// Set Control Mode Label
CASE stat.nCtrlMode	OF
	0:	stat.sCtrlMode	:= 'HHR (Hand-Held Remote)';
	1:	stat.sCtrlMode	:= 'REMOTE';
	2:	stat.sCtrlMode	:= 'SERIAL LINK';
	3:	stat.sCtrlMode	:= 'FIELDBUS';
ELSE
	stat.sCtrlMode	:= 'UNKNOWN';
END_CASE
END_METHOD

END_FUNCTION_BLOCK

// POUs/Pumps/FB_CRYO_PUMP_SERIAL
// Cryo Turbo Molecular Pump Control
FUNCTION_BLOCK FB_CRYO_PUMP_SERIAL EXTENDS FB_CRYO_PUMP_BASE
VAR_INPUT
	{attribute 'OPC.UA.DA' := '0'}
	in_sCmdSuffix:		STRING(16) := '$0D';
	{attribute 'OPC.UA.DA' := '0'}
	in_sReplySuffix:	STRING(16) := '$0D';
END_VAR
VAR_OUTPUT
END_VAR
VAR

	{attribute 'OPC.UA.DA' := '0'}
	comm:		FB_RS_COMM_NO_SIM;			// No simulation yet
	
	// Pointers to structures inside FB_RS_COMM, e.g. ptrCommCfg.
	{attribute 'OPC.UA.DA' := '0'}
	ptrCommCfg:		POINTER TO T_RS_COMM_CFG;	(* Pointer to comm.cfg instance *)
	{attribute 'OPC.UA.DA' := '0'}
	ptrCommCtrl:	POINTER TO T_RS_COMM_CTRL;	(* Pointer to comm.ctrl instance *)
	{attribute 'OPC.UA.DA' := '0'}
	ptrCommStat:	POINTER TO T_RS_COMM_STAT;	(* Pointer to comm.stat instance *)

END_VAR

// Execute the base class object FB_RS_BASE
SUPER^();

METHOD ActivityInitializing
VAR_INPUT
	bExecute:	BOOL;
END_VAR
VAR_INST
	{attribute 'OPC.UA.DA' := '0'}
    nMethodState:	INT := 0;	// State Machine current state
END_VAR
SetAction('ActivityInitializing');


IF NOT bExecute THEN
	nMethodState	:= 0;	// Reset the state machine
	cmdCounter		:= 0;	// Init will start from the first init command after increment
	RETURN;
END_IF

// Handle State Machine
CASE nMethodState OF
	0:	// Set initial state and status
		statRef.bInitialised	:= FALSE;
		statBaseRef.sReply			:= '';
		SetStatus(E_SM_ERROR.OK, 'BUSY');

		nMethodState := 10;				// Go to next state, i.e. INIT_COMM

	10:	// Initialize COMM port
		(* Reset the serial port *)
		ptrCommCtrl^.nCommand	:= E_RS_COMM_CMD.INIT;
		ptrCommCtrl^.bExecute	:= TRUE;

		(* Start the timer by going false/true *)
		fbTimer (IN := FALSE); (* Reset timer *)
		fbTimer (IN := TRUE, PT := T#5S); (* 5 sec timeout for reply *)

		nMethodState 	:= 15;	// On next cycle wait until the comm port is reset, i.e. idle
		
	15:	// Wait IDLE
		fbTimer (IN := TRUE);
		IF comm.stat.nStatus = E_RS_COMM_STATUS.IDLE THEN
			// Communication is IDLE 
			fbTimer (IN := FALSE);	// disable timer 
			statBaseRef.sReply		:= ptrCommStat^.sReply;	// Save the reply

			// TODO Assign the value to a status variable.
			IF NOT M_ReadFromReply(cmdCounter, TRUE)	THEN
				cmdCounter		:= 0;	// Reset command counter
				nMethodState 	:= 10;	// Wait for INIT
			ELSE
				cmdCounter		:= cmdCounter + 1;	// Increment init command index
				fbTimer (IN := FALSE);	// disable timer 
				fbTimer (IN := TRUE, PT := cfgRef.tDelay_Init); // Wait INIT delay
				bCommProblem	:= FALSE;
				nMethodState 	:= 18;	// Execute next device INIT command
			END_IF
		ELSIF comm.stat.nStatus = E_RS_COMM_STATUS.ERROR THEN
			fbTimer (IN := FALSE);
			SetStatus(E_LAKESHORE_ERROR.COMM, 'ERROR: Communication error');	
			bCommProblem	:= TRUE;
			nEvent := E_SM_EVENT.ERRINIT;
			RETURN;
		ELSIF fbTimer.Q THEN
			// Timer expired after 5 sec. This is an error.
			fbTimer (IN := FALSE);
			SetStatus(E_LAKESHORE_ERROR.TIMEOUT, 'ERROR: Communication timeout');	
			bCommProblem	:= TRUE;
			nEvent := E_SM_EVENT.ERRINIT;
			RETURN;
		END_IF

	
	
	18:	// Wait INIT Delay
		fbTimer (IN := TRUE);
		IF fbTimer.Q THEN
			// Timer expired after 5 sec. This is an error.
			fbTimer (IN := FALSE);
			nMethodState 	:= 20;	// Execute next device INIT command
			RETURN;
		END_IF

	
	
	20:	// INIT DEV
		IF ptrInitCmds^ [cmdCounter].cmd = '' THEN
			// Device INIT is done. Go to IDLE 
			statRef.bInitialised 	:= TRUE;
			cmdCounter			:= 1;
			SetStatus(E_SM_ERROR.OK, 'IDLE');
			nEvent 		:= E_SM_EVENT.INITDONE;
			RETURN;
		END_IF
		
		(* Send INIT command with index cmdCounter *)
		ptrCommCtrl^.nCommand		:= E_RS_COMM_CMD.SEND;
		ptrCommCtrl^.sCmd			:= ptrInitCmds^ [cmdCounter].cmd;
		ptrCommCtrl^.nNumReplies	:= 1;
		ptrCommCtrl^.bHasReply		:= TRUE;
		ptrCommCtrl^.bExecute		:= TRUE;
	
		(* Start the timer by going false/true *)
		fbTimer (IN := FALSE); (* Reset timer *)
		fbTimer (IN := TRUE, PT := T#5S); (* 5 sec timeout for reply *)

		// On next cycle wait until the comm port is idle
		nMethodState 	:= 15;	// On next cycle wait until the comm port is idle
	
END_CASE
END_METHOD

METHOD ActivityMonitoring
VAR_INPUT
	bExecute:	BOOL;
END_VAR
VAR_INST
	{attribute 'OPC.UA.DA' := '0'}
    nMethodState:	INT := 0;	// State Machine current state
	{attribute 'OPC.UA.DA' := '0'}
	nRetries:		INT := 0;	// Number of retries in case of communication problems
END_VAR

VAR
	offset: INT;
END_VAR
IF NOT cfgRef.bAutoMonitor AND statRef.nSubstate = E_RS_BASE_SUBSTATE.NOTOP_READY THEN
	SetAction('No Monitoring'); 
	SetStatus(E_SM_ERROR.OK, 'IDLE');
	nMethodState	:= 0;	// Reset the state machine
	cmdCounter		:= 1;	// Reading will start from the first command in the array
	RETURN;
END_IF

IF NOT bExecute THEN
	SetAction('ActivityMonitoring'); 
	SetStatus(E_SM_ERROR.OK, 'BUSY');
	nMethodState	:= 0;	// Reset the state machine
	cmdCounter		:= 1;	// Reading will start from the first command in the array
	RETURN;
END_IF

// Handle State Machine
CASE nMethodState OF
	0:	// Execute a command from the command array
		IF ptrReadCmds^ [cmdCounter].cmd = '' OR cmdCounter > 16 THEN

			// All commands have been executed. 
			// Wait tDelay_Periodic before re-starting the READ.
			cmdCounter	:= 1;
			SetStatus(E_SM_ERROR.OK, 'IDLE');
			
			(* Start the timer by going false/true *)
			fbTimer (IN := FALSE); (* Reset timer *)
			fbTimer (IN := TRUE, PT := cfgRef.tDelay_Periodic);
			nMethodState := 10;				// Goto Wait for tDelay_Periodic
			RETURN;
			
		END_IF
		
		(* Send command with index cmdCounter *)
		ptrCommCtrl^.nCommand		:= E_RS_COMM_CMD.SEND;
		ptrCommCtrl^.sCmd			:= ptrReadCmds^ [cmdCounter].cmd;
		ptrCommCtrl^.nNumReplies	:= 1;
		ptrCommCtrl^.bHasReply		:= TRUE;
		ptrCommCtrl^.bExecute		:= TRUE;
		
		// In case we are executing 'SET' commands, there are no replies.
		// However, we need a delay of at least 50ms between commands.
		// We will apply 150ms.
		IF NOT ptrCommCtrl^.bHasReply THEN
			// There is no reply, i.e. this is a 'SET' command.
			// Start the timer by going false/true.
			// Apply 200ms delay between SET commands.
			fbTimer (IN := FALSE); // Reset timer
			fbTimer (IN := TRUE, PT := T#200MS); 
			cmdCounter		:= cmdCounter + 1;	// Go to next command.
			nMethodState	:= 10;				// Goto WAIT for Reading to complete,
			RETURN;
		ELSE			
			// There is a reply, i.e. this is a 'READ' command.
			// Apply short delay of 10ms before checking the status. 
			// Start the timer by going false/true
			fbTimer (IN := FALSE); // Reset timer
			fbTimer (IN := TRUE, PT := T#10MS);	
			statRef.sErrorText	:= 'BUSY';
			nMethodState := 15;	// Goto WAIT for Reading to complete,
		END_IF
		

	10:	// Wait until the delay timeout expires
		fbTimer (IN := TRUE);

		(* If Timer has expired, go to the next state. *)
		IF fbTimer.Q THEN
			fbTimer (IN := FALSE);
			nMethodState 	:= 0;	// Goto Wait for tDelay_Periodic
			RETURN;
		END_IF
	
	15:	// Wait until the delay timeout expires
		fbTimer (IN := TRUE);

		(* If Timer has expired, go to the next state. *)
		IF fbTimer.Q THEN
			fbTimer (IN := FALSE);
			fbTimer (IN := TRUE, PT := T#5S);	// 5 sec timeout for reply
			statRef.sErrorText	:= 'BUSY';
			nMethodState 	:= 20;	// Goto Wait for IDLE/Reply
			RETURN;
		END_IF
	



	20:	// Wait for the reading to complete, i.e. IDLE
		fbTimer (IN := TRUE);
		IF comm.stat.nStatus = E_RS_COMM_STATUS.IDLE THEN
			// Communication is IDLE 
			fbTimer (IN := FALSE);	// disable timer 
			statBaseRef.sReply		:= ptrCommStat^.sReply;	// Save the reply
			
			// Copy readings to status variable(s)
			
			// TODO Assign the value to a status variable.
			IF NOT M_ReadFromReply(cmdCounter, FALSE)	THEN
				// Reply was not OK. Maybe out of sync.
				// Re-INIT the communication, i.e. clear the buffer.
				ptrCommCtrl^.nCommand	:= E_RS_COMM_CMD.INIT;
				ptrCommCtrl^.bExecute	:= TRUE;
		
				(* Start the timer by going false/true *)
				fbTimer (IN := FALSE); (* Reset timer *)
				fbTimer (IN := TRUE, PT := T#5S); (* 5 sec timeout for reply *)
		
				SetStatus(E_LAKESHORE_ERROR.COMM, 'ERROR: Communication error');	
				bCommProblem	:= TRUE;

				nMethodState 	:= 10;	// On next cycle wait until the comm port is reset, i.e. idle
				RETURN;
			ELSE
				// All OK. Go to next command.
				bCommProblem	:= FALSE;
				nRetries		:= 0;	// Reset number of retries
		
				cmdCounter		:= cmdCounter + 1;	// Go to next command.
				
				// Apply a 50 ms delay between commands
				fbTimer (IN := FALSE);	// Reset timer
				fbTimer (IN := TRUE, PT := T#50MS); 
				nMethodState := 10;		// Apply delay
				nEvent := E_SM_EVENT.COMMOK;
				RETURN;
			END_IF
		ELSIF comm.stat.nStatus = E_RS_COMM_STATUS.ERROR OR fbTimer.Q THEN
			// No Reply.
			// Re-INIT the communication, i.e. clear the buffer.
			ptrCommCtrl^.nCommand	:= E_RS_COMM_CMD.INIT;
			ptrCommCtrl^.bExecute	:= TRUE;
	
			(* Start the timer by going false/true *)
			fbTimer (IN := FALSE); (* Reset timer *)
			fbTimer (IN := TRUE, PT := T#5S); (* 5 sec timeout for reply *)
	
			SetStatus(E_LAKESHORE_ERROR.COMM, 'ERROR: Communication error');	
			bCommProblem	:= TRUE;

			nRetries		:= nRetries + 1;		// Increment number of retries
			statBaseRef.nRetries	:= statBaseRef.nRetries + 1;	// Increment total number of retries

			nMethodState 	:= 10;	// On next cycle wait until the comm port is reset, i.e. idle
			RETURN;
		END_IF

	
END_CASE
END_METHOD

METHOD M_ExecuteComm
VAR_INPUT
END_VAR
comm(in_sCmdSuffix:=in_sCmdSuffix, in_sReplySuffix:=in_sReplySuffix, in_nTimeout:=3000);
END_METHOD

METHOD M_GetCouplerState : BOOL
VAR_INPUT
END_VAR
IF comm.i_nCouplerState = 8 THEN
	M_GetCouplerState	:= TRUE;	
ELSE
	M_GetCouplerState	:= FALSE;	
END_IF
END_METHOD

// Add checksum at the end of Pfeiffer Vacuum Protocol (PVP) command
METHOD M_PVP_Checksum : STRING(24)
VAR_INPUT
	sCmd:	STRING;	// Command without the checksum
END_VAR
VAR
	i:			INT;
	nVar:		SINT;
	nSum:		INT;
	nRes:		INT;	// Resulting check sum
	sCmdFull:	STRING(24);	// Command with the checksum
    fbFormat:	FB_FormatString;
	sTmp:		T_MaxString;
	length:		INT;
END_VAR
// Get the command length
length	:= LEN(sCmd);

nSum	:= 0;
FOR i:=0 TO (length-1) DO
	nSum	:= nSum + BYTE_TO_SINT(sCmd[i]);
END_FOR
nRes	:= nSum MOD 256;

sTmp	:= sCmd;
fbFormat(	sFormat := '%s%.3d', 
			arg1 := F_STRING(sTmp), 
			arg2 := F_INT(nRes), 
			sOut => sCmdFull);
			
M_PVP_Checksum	:= sCmdFull;
END_METHOD

METHOD M_ReadFromReply : BOOL
// Method to check correctness of the reply and assign the result to a status variable.
VAR_INPUT
	idx:		INT;		(* arr [idx] will hold the first extracted value, arr [idx+1] the second one, etc. *)
	bInitCmd:	BOOL := FALSE;
END_VAR
VAR
	pos:	INT;
	cmd:	STRING;
	length:	DINT;
	subStr:	STRING(255);
END_VAR
// TODO: Implement specific parsing of replies
END_METHOD

END_FUNCTION_BLOCK

// POUs/Pumps/FB_CRYO_PUMP_ECODRY
FUNCTION_BLOCK FB_CRYO_PUMP_ECODRY EXTENDS FB_CRYO_PUMP_MODBUS
VAR_INPUT
END_VAR
VAR_OUTPUT
END_VAR
VAR CONSTANT
END_VAR
VAR
	{attribute 'OPC.UA.DA' := '1'}
	cfg:		T_CRYO_PUMP_MODBUS_CFG;		//  Config parameters
	{attribute 'OPC.UA.DA' := '1'}
	ctrl:		T_CRYO_PUMP_MODBUS_CTRL;	//  Control parameters
	{attribute 'OPC.UA.DA' := '1'}
	{attribute 'OPC.UA.DA.Access' := '1'}
	stat:		T_CRYO_PUMP_MODBUS_STAT;	//  Status parameters - ReadOnly


END_VAR

// Execute the base class object FB_RS_BASE
SUPER^();

METHOD M_Configure
VAR_INPUT
END_VAR
IF NOT bStarted	THEN
	//
	// START: Mandatory for ALL pumps !!!
	//
	// Set references from FB_RS_BASE
	cfgRef	REF=cfg;
	ctrlRef	REF=ctrl;
	statRef	REF=stat;

	// Set references from FB_CRYO_PUMP_BASE
	cfgBaseRef	REF=cfg;
	ctrlBaseRef	REF=ctrl;
	statBaseRef	REF=stat;

	// Set references from FB_CRYO_PUMP_MODBUS
	cfgModbusRef	REF=cfg;
	ctrlModbusRef	REF=ctrl;
	statModbusRef	REF=stat;

	// Copy input parameters to configuration
	cfg.nModel			:= in_nModel;
	cfg.bAutoMonitor	:= in_bAutoMonitor;
	cfg.tDelay_Periodic	:= DINT_TO_TIME(in_nPeriod);
	
	
	// Set pointers to arrays of commands
//	ptrInitCmds	:= ADR(cfg.cmdList_Init);(* Pointer to INIT commands *)
//	ptrReadCmds	:= ADR(cfg.cmdList_Read);(* Pointer to READ commands *)
	
	// TODO in FB that extends the functionality
	// Set pointers to comm, i.e.
	ptrCommCfg	:= ADR(comm.cfg);	(* Pointer to comm.cfg instance *)
	ptrCommCtrl	:= ADR(comm.ctrl);	(* Pointer to comm.ctrl instance *)
	ptrCommStat	:= ADR(comm.stat);	(* Pointer to comm.stat instance *)
	
	// Set comm suffixes for commands and replies
//	ptrCommCfg^.sCmdSuffix		:= '';
//	ptrCommCfg^.sReplySuffix	:= '';

	statRef.bConfigured	:= TRUE;
	bStarted			:= TRUE;
	//
	// END: Mandatory for ALL pumps !!!
	//


	// TODO USER
	// Add here real configuration
	IF in_sVersion = 'V01'	THEN
		cfg.nVersion	:= E_ECODRY_VERSION.V01;
	ELSIF in_sVersion = 'V21'  OR  in_sVersion = 'V22'	THEN
		cfg.nVersion	:= E_ECODRY_VERSION.V21_22;
	END_IF
	
	// Adjust addresses and number of words
	CASE cfg.nVersion	OF
		E_ECODRY_VERSION.V01:
			// Set register addresses
			cfg.aAddr [1]	:= 16#0040;
			cfg.aAddr [2]	:= 16#0067;
			cfg.aAddr [3]	:= 16#0667;
			cfg.aAddr [4]	:= 0;	// Unused address must be zero
			
			// Set number of words to read
			cfg.aWords [1]	:= 16;
			cfg.aWords [2]	:= 2;
			cfg.aWords [3]	:= 6;
			cfg.aWords [4]	:= 0;	// Number of words for unused address must be zero
	END_CASE
	
	cfg.nSlaveID	:= in_nSlaveID;

	
END_IF
END_METHOD

METHOD M_ExtractReadings_V01 : BOOL
VAR_INPUT
	nAddressIndex:	INT;	// Which address space to read
END_VAR
VAR
	pBuf:	POINTER TO BYTE	:= ADR(stat.nInputBuffer);
	loop:	INT;
	par:	INT;
END_VAR
// There are 3 bytes before data starts !!!
IF nAddressIndex = 1 THEN
	////////////////////////////
	// Extract Common Parameters
	////////////////////////////

	// Reference Frequency 0x40H
	// Offset 3 + 0 = 3
	stat.lrFreqRef		:= UINT_TO_LREAL(M_ByteSwapUINT(ADR(pBuf[3]))) / 100.0;
	stat.lrOutFreq		:= INT_TO_LREAL(M_ByteSwapINT(ADR(pBuf[5]))) / 100.0;
	stat.nPumpSpeed		:= LREAL_TO_DINT(stat.lrOutFreq * 60.0);	// [Hz] -> [rpm]
	stat.nMotorCurr		:= UINT_TO_DINT(M_ByteSwapUINT(ADR(pBuf[7]))) * 10;
	stat.lrOutVoltRef	:= UINT_TO_LREAL(M_ByteSwapUINT(ADR(pBuf[13]))) / 10.0;
	stat.nMotorVolt		:= UINT_TO_DINT(M_ByteSwapUINT(ADR(pBuf[15])));
	stat.lrOutPower		:= INT_TO_LREAL(M_ByteSwapINT(ADR(pBuf[17]))) / 10.0;
	
	stat.nOpTime	:= M_ByteSwapUINT(ADR(pBuf[27]));
	stat.nSwFlash	:= M_ByteSwapUINT(ADR(pBuf[29]));

	(*
	stat.lrTemperature	:= UINT_TO_LREAL(M_ByteSwapUINT(ADR(pBuf[83])));

	stat.nSwRom		:= M_ByteSwapUINT(ADR(pBuf[57]));
	stat.nNumRunCmd	:= M_ByteSwapUINT(ADR(pBuf[109]));
	stat.nFanOpTime	:= M_ByteSwapUINT(ADR(pBuf[81]));
	*)

ELSIF nAddressIndex = 2 THEN
	stat.nFanOpTime			:= M_ByteSwapUINT(ADR(pBuf[3]));
	stat.nElecTemp			:= UINT_TO_DINT(M_ByteSwapUINT(ADR(pBuf[5])));
ELSIF nAddressIndex = 3 THEN
	stat.nServiceHours		:= M_ByteSwapUINT(ADR(pBuf[3]));
	stat.nNumPumpDowns		:= M_ByteSwapUINT(ADR(pBuf[7]));
	stat.nDaysUntilService	:= M_ByteSwapUINT(ADR(pBuf[13]));
END_IF
END_METHOD

METHOD M_ExtractReadings_V21_22 : BOOL
VAR_INPUT
	nAddressIndex:	INT;	// Which address space to read
END_VAR
VAR
	pBuf:	POINTER TO BYTE	:= ADR(stat.nInputBuffer);
	loop:	INT;
	par:	INT;
END_VAR
// There are 3 bytes before data starts !!!
IF nAddressIndex = 1 THEN
	////////////////////////////
	// Extract Common Parameters
	////////////////////////////

	// Reference Frequency 0x40H
	// Offset 3 + 0 = 3
	stat.lrFreqRef		:= UINT_TO_LREAL(M_ByteSwapUINT(ADR(pBuf[3]))) / 100.0;
	stat.lrOutFreq		:= INT_TO_LREAL(M_ByteSwapINT(ADR(pBuf[5]))) / 100.0;
	stat.nMotorCurr		:= UINT_TO_DINT(M_ByteSwapUINT(ADR(pBuf[7]))) * 10;
	stat.lrOutVoltRef	:= UINT_TO_LREAL(M_ByteSwapUINT(ADR(pBuf[13]))) / 10.0;
	stat.nMotorVolt		:= UINT_TO_DINT(M_ByteSwapUINT(ADR(pBuf[15])));
	stat.lrOutPower		:= INT_TO_LREAL(M_ByteSwapINT(ADR(pBuf[17]))) / 10.0;
	
	stat.nOpTime	:= M_ByteSwapUINT(ADR(pBuf[27]));
	stat.nSwFlash	:= M_ByteSwapUINT(ADR(pBuf[29]));

	(*
	stat.lrTemperature	:= UINT_TO_LREAL(M_ByteSwapUINT(ADR(pBuf[83])));

	stat.nSwRom		:= M_ByteSwapUINT(ADR(pBuf[57]));
	stat.nNumRunCmd	:= M_ByteSwapUINT(ADR(pBuf[109]));
	stat.nFanOpTime	:= M_ByteSwapUINT(ADR(pBuf[81]));
	*)

ELSIF nAddressIndex = 2 THEN
	stat.nFanOpTime			:= M_ByteSwapUINT(ADR(pBuf[3]));
	stat.nElecTemp			:= UINT_TO_DINT(M_ByteSwapUINT(ADR(pBuf[5])));
ELSIF nAddressIndex = 3 THEN
	stat.nServiceHours		:= M_ByteSwapUINT(ADR(pBuf[3]));
	stat.nNumPumpDowns		:= M_ByteSwapUINT(ADR(pBuf[7]));
	stat.nDaysUntilService	:= M_ByteSwapUINT(ADR(pBuf[13]));
END_IF
END_METHOD

METHOD M_IsReady : BOOL
VAR_INPUT
END_VAR
//	M_UpdateStatus() sets the stat.bReady flag.
M_IsReady	:= stat.bReady;
END_METHOD

METHOD M_IsRunning : BOOL
VAR_INPUT
END_VAR
M_IsRunning	:= stat.bReady OR stat.nPumpSpeed > 0;
END_METHOD

METHOD M_ReadFromReply : BOOL
VAR_INPUT
	nAddressIndex:	INT;	// Which address space to read
END_VAR
IF cfg.nVersion	= E_ECODRY_VERSION.V01	THEN
	M_ExtractReadings_V01    (nAddressIndex);
ELSIF cfg.nVersion	= E_ECODRY_VERSION.V21_22	THEN
	M_ExtractReadings_V21_22 (nAddressIndex);
END_IF
END_METHOD

METHOD M_UpdateStatus
VAR_INPUT
END_VAR
// Update inputs
stat.bReady		:= NOT i_bRunning;	// Active low
END_METHOD

END_FUNCTION_BLOCK

// POUs/Pumps/FB_CRYO_PUMP_MODBUS
FUNCTION_BLOCK FB_CRYO_PUMP_MODBUS EXTENDS FB_CRYO_PUMP_BASE
VAR_INPUT
	{attribute 'OPC.UA.DA' := '0'}
	in_nSlaveID:	BYTE := 1;		// Slave ID
	{attribute 'OPC.UA.DA' := '0'}
	in_sVersion:	STRING := 'V21';	// Version number. String starting with 'V', e.g. 'V21'.
END_VAR
VAR_OUTPUT
END_VAR
VAR CONSTANT
END_VAR
VAR
	{attribute 'OPC.UA.DA' := '0'}
	cfgModbusRef:	REFERENCE TO T_CRYO_PUMP_MODBUS_CFG;
	{attribute 'OPC.UA.DA' := '0'}
	ctrlModbusRef:	REFERENCE TO T_CRYO_PUMP_MODBUS_CTRL;
	{attribute 'OPC.UA.DA' := '0'}
	statModbusRef:	REFERENCE TO T_CRYO_PUMP_MODBUS_STAT;
	
	{attribute 'OPC.UA.DA' := '0'}
	comm:		FB_MODBUS_COMM_NO_SIM;		// Instance of generic comm object. OPC UA Disabled!!!
	
	(* Pointers *)
	{attribute 'OPC.UA.DA' := '0'}
	ptrCommCfg:		POINTER TO T_MODBUS_CFG 	:= ADR(comm.cfg);	(* Pointer to comm.cfg instance *)
	{attribute 'OPC.UA.DA' := '0'}
	ptrCommCtrl:	POINTER TO T_MODBUS_CTRL 	:= ADR(comm.ctrl);	(* Pointer to comm.ctrl instance *)
	{attribute 'OPC.UA.DA' := '0'}
	ptrCommStat:	POINTER TO T_MODBUS_STAT 	:= ADR(comm.stat);	(* Pointer to comm.stat instance *)


	(* Timers *)


	// Input signals
	i_bRunning		AT %I*:	BOOL;	// TRUE, if pump is running


END_VAR

// Execute the base class object FB_CRYO_PUMP_BASE
SUPER^();

METHOD ActivityInitializing
VAR_INPUT
	bExecute:	BOOL;
END_VAR
VAR_INST
	{attribute 'OPC.UA.DA' := '0'}
    nMethodState:	INT := 0;	// State Machine current state
END_VAR
VAR
	nInt:	INT;	// Temporary INT for conversion of ENUM types
END_VAR
SetAction('ActivityInitializing');


IF NOT bExecute THEN
	nMethodState	:= 0;	// Reset the state machine
	RETURN;
END_IF

// Handle State Machine
CASE nMethodState OF
	0:	// Set communication parameters and Model configuration


		// Set monitoring period (input parameter)
		cfgRef.tDelay_Periodic	:= DINT_TO_TIME(in_nPeriod);
		// Auto monitor, i.e. monitor in Standby_Ready as well
		cfgRef.bAutoMonitor	:= TRUE;

		(* Set initial state and status *)
		statRef.bInitialised	:= FALSE;
		statBaseRef.nRetries		:= 0;

		SetStatus(E_SM_ERROR.OK, 'BUSY');
		
		// User configuration of the system
//		M_UserConfigure();

		nMethodState := 10;				// Go to next state, i.e. INIT_COMM

	10:	// Initialize COMM port
		(* Reset the serial port *)
		nInt	:= E_RS_COMM_CMD.INIT;
		ptrCommCtrl^.nCommand	:= nInt;
		ptrCommCtrl^.bExecute	:= TRUE;

		(* Start the timer by going false/true *)
		fbTimer (IN := FALSE); (* Reset timer *)
		fbTimer (IN := TRUE, PT := T#5S); (* 5 sec timeout for reply *)

		nMethodState 	:= 15;	// On next cycle wait until the comm port is reset, i.e. idle
		
	15:	// Wait IDLE
		fbTimer (IN := TRUE);
		IF comm.stat.nStatus = E_RS_COMM_STATUS.IDLE THEN
			// Communication is IDLE 
			fbTimer (IN := FALSE);	// disable timer 
			statModbusRef.nInputBuffer		:= ptrCommStat^.DeviceReply;	// Save the reply

			bCommProblem	:= FALSE;
			// Device INIT is done. Go to IDLE 
			statRef.bInitialised 	:= TRUE;
			SetStatus(E_CCC_STATUS.IDLE, 'IDLE');
			nEvent 		:= E_SM_EVENT.INITDONE;
			RETURN;
		ELSIF comm.stat.nStatus = E_RS_COMM_STATUS.ERROR THEN
			fbTimer (IN := FALSE);
			SetStatus(E_CCC_ERROR.COMM, 'ERROR: Communication error');	
			bCommProblem	:= TRUE;
			nEvent := E_SM_EVENT.ERRINIT;
			RETURN;
		ELSIF fbTimer.Q THEN
			// Timer expired after 5 sec. This is an error.
			fbTimer (IN := FALSE);
			SetStatus(E_CCC_ERROR.TIMEOUT, 'ERROR: Communication timeout');	
			bCommProblem	:= TRUE;
			nEvent := E_SM_EVENT.ERRINIT;
			RETURN;
		END_IF

	
	
	
END_CASE
END_METHOD

METHOD ActivityMonitoring
VAR_INPUT
	bExecute:	BOOL;
END_VAR
VAR_INST
	{attribute 'OPC.UA.DA' := '0'}
    nMethodState:	INT := 0;			// State Machine current state
	{attribute 'OPC.UA.DA' := '0'}
	nAddressIndex:	INT := 1;			// Which address space to read
	{attribute 'OPC.UA.DA' := '0'}
	nRetries:		INT := 0;			// Number of retries in case of communication problems
END_VAR
IF NOT bExecute THEN
	SetAction('ActivityMonitoring'); 
	SetStatus(E_SM_ERROR.OK, 'BUSY');
	nMethodState	:= 0;	// Reset the state machine
	nAddressIndex	:= 1;
	ctrlModbusRef.nRegister	:= cfgModbusRef.aAddr  [1];
	ctrlModbusRef.nWords	:= cfgModbusRef.aWords [1];
	nRetries		:= 0;					
	RETURN;
END_IF

// Handle State Machine
CASE nMethodState OF
	0:	// Execute a command from the command array
		// Check if we have to exit Monitoring
		IF nNextState <> E_RS_BASE_STATE.NONE	THEN
			SetStatus(E_SM_ERROR.OK, nNextDescription);
			SetState(nNextState, nNextSubstate);
			nNextState		:= E_RS_BASE_STATE.NONE;
			nNextSubstate	:= E_RS_BASE_SUBSTATE.NONE;
			nNextDescription:= 'IDLE';
			RETURN;
		END_IF
		
		
		// Send command
		ptrCommCtrl^.nCommand		:= E_MODBUS_CMD.SEND;
		ptrCommCtrl^.nSlaveID		:= cfgModbusRef.nSlaveID;
		ptrCommCtrl^.nRegister		:= ctrlModbusRef.nRegister;
		ptrCommCtrl^.nWords			:= ctrlModbusRef.nWords;
		ptrCommCtrl^.bExecute		:= TRUE;
		
		(* Start the timer by going false/true *)
		fbTimer (IN := FALSE); (* Reset timer *)
		fbTimer (IN := TRUE, PT := T#5S); (* 5 sec timeout for reply *)

		nMethodState := 20;				// Goto WAIT for Reading to complete,

	10:	// Wait until the delay timeout expires
		fbTimer (IN := TRUE);

		// Check if we have to exit Monitoring
		IF nNextState <> E_RS_BASE_STATE.NONE THEN
			fbTimer (IN := FALSE); (* Stop the timer *)
			SetStatus(E_SM_ERROR.OK, nNextDescription);
			SetState(nNextState, nNextSubstate);
			nNextState		:= E_RS_BASE_STATE.NONE;
			nNextSubstate	:= E_RS_BASE_SUBSTATE.NONE;
			nNextDescription:= 'IDLE';
			RETURN;
		END_IF
	
		(* If Timer has expired, go to the next state. *)
		IF fbTimer.Q THEN
			fbTimer (IN := FALSE);
			SetStatus(E_SM_ERROR.OK, 'BUSY');
			nMethodState 	:= 0;	// Goto next reading
			RETURN;
		END_IF
	


	20:	// Wait for the reading to complete, i.e. IDLE
		fbTimer (IN := TRUE);
		IF comm.stat.nStatus = E_RS_COMM_STATUS.IDLE THEN
			// Communication is IDLE  
			fbTimer (IN := FALSE);	// disable timer 
			statModbusRef.nInputBuffer		:= ptrCommStat^.DeviceReply;	// Save the reply
			
			// Extract the readings from the reply.
			M_ReadFromReply(nAddressIndex);

			bCommProblem	:= FALSE;
			nRetries		:= 0;	// Reset number of retries
			
			// Check if we have to exit Monitoring
			IF nNextState <> E_RS_BASE_STATE.NONE THEN
				fbTimer (IN := FALSE); (* Stop the timer *)
				SetStatus(E_SM_ERROR.OK, nNextDescription);
				SetState(nNextState, nNextSubstate);
				nNextState		:= E_RS_BASE_STATE.NONE;
				nNextSubstate	:= E_RS_BASE_SUBSTATE.NONE;
				nNextDescription:= 'IDLE';
				RETURN;
			END_IF
	
			IF NOT M_SetCommand(nAddressIndex) THEN
				// We completed a full read cycle.
				// Wait periodic delay.
				// Periodic READ is done. Wait tDelay_Periodic before re-starting the READ.
				SetStatus(E_SM_ERROR.OK, 'IDLE');
				(* Start the timer by going false/true *)
				fbTimer (IN := FALSE); (* Reset timer *)
				fbTimer (IN := TRUE, PT := cfgRef.tDelay_Periodic);
				nMethodState := 10;				// Goto Wait 
				RETURN;
			ELSE
				// Apply a short delay of 30 ms after each command
				fbTimer (IN := FALSE); (* Reset timer *)
				fbTimer (IN := TRUE, PT := T#30MS);
				nMethodState := 10;				// Goto Wait 
				RETURN;
			END_IF

		ELSIF INT_TO_DINT(comm.stat.nStatus) = INT_TO_DINT(E_MODBUS_STATUS.ERROR) OR fbTimer.Q THEN
			fbTimer (IN := FALSE);
			SetStatus(E_MODBUS_ERROR.RECEIVE, 'ERROR: Communication error');	
			bCommProblem	:= TRUE;
			// Retry up to 3 times
			nRetries		:= nRetries + 1;		// Increment number of retries
			statModbusRef.nRetries	:= statModbusRef.nRetries + 1;	// Increment total number of retries
			IF nRetries > 3 THEN
				nEvent := E_SM_EVENT.ERRCOMM;
			ELSE
				// Apply a short delay of 1 sec and retry
				fbTimer (IN := FALSE); (* Reset timer *)
				fbTimer (IN := TRUE, PT := T#1000MS);
				nMethodState := 10;				// Goto Wait 
			END_IF
			RETURN;
		END_IF

	
END_CASE
END_METHOD

METHOD M_ByteSwapFLOAT : REAL
VAR_INPUT
	pByte:		POINTER TO BYTE;	// Pointer to array of bytes read from JUMO
END_VAR
VAR
	rResult:	REAL;
	pResult:	POINTER TO BYTE	:= ADR(rResult);	// Pointer to the result
END_VAR
pResult[0]	:= pByte[1];
pResult[1]	:= pByte[0];
pResult[2]	:= pByte[3];
pResult[3]	:= pByte[2];

M_ByteSwapFLOAT	:= rResult;
END_METHOD

METHOD M_ByteSwapINT : INT
VAR_INPUT
	pByte:		POINTER TO BYTE;	// Pointer to array of bytes read from JUMO
END_VAR
VAR
	nResult:	INT;
	pResult:	POINTER TO BYTE	:= ADR(nResult);	// Pointer to the result
END_VAR
pResult[0]	:= pByte[1];
pResult[1]	:= pByte[0];

M_ByteSwapINT	:= nResult;
END_METHOD

METHOD M_ByteSwapUINT : UINT
VAR_INPUT
	pByte:		POINTER TO BYTE;	// Pointer to array of bytes read from JUMO
END_VAR
VAR
	nResult:	UINT;
	pResult:	POINTER TO BYTE	:= ADR(nResult);	// Pointer to the result
END_VAR
pResult[0]	:= pByte[1];
pResult[1]	:= pByte[0];

M_ByteSwapUINT	:= nResult;
END_METHOD

METHOD M_ExecuteComm
VAR_INPUT
END_VAR
(* Execute comm instance *)
comm(	in_bSimulation	:= in_bSimulation,
		in_nModel		:= 0,
		in_cReadFunction:= 3);
END_METHOD

METHOD M_GetCouplerState : BOOL
VAR_INPUT
END_VAR
IF comm.i_nCouplerState = 8 THEN
	M_GetCouplerState	:= TRUE;	
ELSE
	M_GetCouplerState	:= FALSE;	
END_IF
END_METHOD

METHOD M_ReadFromReply : BOOL
VAR_INPUT
	nAddressIndex:	INT;	// Which address space to read
END_VAR
// TODO: For every pump implementation
END_METHOD

METHOD M_SetCommand : BOOL
VAR_IN_OUT
	nAddressIndex:	INT;	// Which address space to read
END_VAR
// We always read from ECODRY
ctrlModbusRef.nCmdType	:= E_MODBUS_CMD_TYPE.READ;

// Go to next register address to read
nAddressIndex	:= nAddressIndex + 1;

IF nAddressIndex > 8  OR  cfgModbusRef.aAddr[nAddressIndex] = 0	OR  cfgModbusRef.aWords[nAddressIndex] = 0	THEN
	ctrlModbusRef.nRegister	:= cfgModbusRef.aAddr  [1];
	ctrlModbusRef.nWords	:= cfgModbusRef.aWords [1];
	nAddressIndex	:= 1;
	M_SetCommand	:= FALSE;	// Restarting from first address
ELSE
	ctrlModbusRef.nRegister	:= cfgModbusRef.aAddr  [nAddressIndex];
	ctrlModbusRef.nWords	:= cfgModbusRef.aWords [nAddressIndex];
	M_SetCommand	:= TRUE;	
END_IF
END_METHOD

END_FUNCTION_BLOCK

// POUs/Pumps/FB_CRYO_PUMP_HIPACE30
FUNCTION_BLOCK FB_CRYO_PUMP_HIPACE30 EXTENDS FB_CRYO_PUMP_SERIAL
VAR_INPUT
END_VAR
VAR_OUTPUT
END_VAR
VAR
	
	{attribute 'OPC.UA.DA' := '1'}
	cfg:		T_CRYO_PUMP_HIPACE30_CFG;	
	{attribute 'OPC.UA.DA' := '1'}
	ctrl:		T_CRYO_PUMP_BASE_CTRL;	
	{attribute 'OPC.UA.DA' := '1'}
	{attribute 'OPC.UA.DA.Access' := '1'}
	stat:		T_CRYO_PUMP_HIPACE30_STAT;	


	// Input signals
	i_bReady		AT %I*:	BOOL;	// Turbo Pump Ready (signal DO1)
	i_bError		AT %I*:	BOOL;	// If FALSE, Error present - active low (signal DO2)

	// Output signals q_bStart already defined in FB_CRYO_TMP_BASE.
	// q_bStart should activate a relay that 
	// connects Pin 7 with Pin 5 - DI Pumping station

END_VAR


// Execute the base class object FB_CRYO_PUMP_SERIAL
SUPER^();

METHOD M_Configure
VAR_INPUT
END_VAR
VAR
	//
	// List of INIT commands.
	//
	cmdList_Init_HIPACE30:	ARRAY [1..8] OF T_CRYO_PUMP_CMD := [
		(cmd := cfg.C_CMD_sCtrlViaInt, 		length := 17),	// Reply of 17 chars with the terminator!	
		(cmd := cfg.C_CMD_sFwVersion, 		length := 20),	
		(cmd := cfg.C_CMD_sHwVersion, 		length := 20),
		(cmd := cfg.C_CMD_nNominalSpeed,	length := 20),
		(cmd := '', 						length := 0),
		(cmd := '', 						length := 0),
		(cmd := '', 						length := 0),
		(cmd := '', 						length := 0)];

	//
	//	List of READ (and WRITE) commands.
	// NOTE: Monitoring loop stops on first cmd = ''.
	//
	cmdList_Read_HIPACE30:	ARRAY [1..16] OF T_CRYO_PUMP_CMD := [
		(cmd := cfg.C_CMD_bON, 				length := 20),	// 20 chars with the terminator!	
		(cmd := cfg.C_CMD_nCtrlMode, 		length := 17),	
		(cmd := cfg.C_CMD_sErrorCode, 		length := 20),
		(cmd := cfg.C_CMD_bTargetSpeed, 	length := 20),
		(cmd := cfg.C_CMD_nMotorCurr, 		length := 20),
		(cmd := cfg.C_CMD_nPumpHours, 		length := 20),
		(cmd := cfg.C_CMD_nMotorVolt, 		length := 20),
		(cmd := cfg.C_CMD_nElecHours, 		length := 20),
		(cmd := cfg.C_CMD_nElecTemp, 		length := 20),
		(cmd := cfg.C_CMD_nPumpTemp, 		length := 20),
		(cmd := cfg.C_CMD_nPumpSpeed, 		length := 20),
		(cmd := '', 						length := 0),
		(cmd := '', 						length := 0),
		(cmd := '', 						length := 0),
		(cmd := '', 						length := 0),
		(cmd := '', 						length := 0)];
	
		i:	INT;
END_VAR
IF NOT bStarted	THEN
	//
	// START: Mandatory for ALL pumps !!!
	//
	// Set references from FB_RS_BASE
	cfgRef	REF=cfg;
	ctrlRef	REF=ctrl;
	statRef	REF=stat;

	// Set references from FB_CRYO_TMP_BASE
	cfgBaseRef	REF=cfg;
	ctrlBaseRef	REF=ctrl;
	statBaseRef	REF=stat;
	
	// Copy input parameters to configuration
	cfg.nModel			:= in_nModel;
	cfg.bAutoMonitor	:= in_bAutoMonitor;
	cfg.tDelay_Periodic	:= DINT_TO_TIME(in_nPeriod);
	
	
	// Set pointers to arrays of commands
	ptrInitCmds	:= ADR(cfg.cmdList_Init);(* Pointer to INIT commands *)
	ptrReadCmds	:= ADR(cfg.cmdList_Read);(* Pointer to READ commands *)
	
	// TODO in FB that extends the functionality
	// Set pointers to comm, i.e.
	ptrCommCfg	:= ADR(comm.cfg);	(* Pointer to comm.cfg instance *)
	ptrCommCtrl	:= ADR(comm.ctrl);	(* Pointer to comm.ctrl instance *)
	ptrCommStat	:= ADR(comm.stat);	(* Pointer to comm.stat instance *)
	
	// Set comm suffixes for commands and replies
	ptrCommCfg^.sCmdSuffix		:= in_sCmdSuffix;
	ptrCommCfg^.sReplySuffix	:= in_sReplySuffix;

	statRef.bConfigured	:= TRUE;
	bStarted			:= TRUE;
	//
	// END: Mandatory for ALL pumps !!!
	//


	//
	// ATH specific configuration
	//
	
	// Assign INIT and READ commands.
	cfg.cmdList_Init	:= cmdList_Init_HIPACE30;
	cfg.cmdList_Read	:= cmdList_Read_HIPACE30;
	
	// Add checksum to all INIT and READ commands
	FOR i:=1 TO 8 DO
		IF cfg.cmdList_Init[i].cmd <> '' THEN
			cfg.cmdList_Init[i].cmd	:= M_PVP_Checksum(cfg.cmdList_Init[i].cmd);
		ELSE
			EXIT;
		END_IF
	END_FOR
	
	FOR i:=1 TO 16 DO
		IF cfg.cmdList_Read[i].cmd <> '' THEN
			cfg.cmdList_Read[i].cmd	:= M_PVP_Checksum(cfg.cmdList_Read[i].cmd);
		ELSE
			EXIT;
		END_IF
	END_FOR
	
END_IF
END_METHOD

METHOD M_GetSpeed : DINT
VAR_INPUT
END_VAR
M_GetSpeed	:= stat.nPumpSpeed;
END_METHOD

METHOD M_IsReady : BOOL
VAR_INPUT
END_VAR
M_IsReady	:= stat.bReady;
END_METHOD

METHOD M_IsRunning : BOOL
VAR_INPUT
END_VAR
M_IsRunning	:= stat.bMoving;
END_METHOD

METHOD M_ReadFromReply : BOOL
// Method to check correctness of the reply and assign the result to a status variable.
VAR_INPUT
	idx:		INT;		(* arr [idx] will hold the first extracted value, arr [idx+1] the second one, etc. *)
	bInitCmd:	BOOL := FALSE;
END_VAR
VAR
	pos:	INT;
	cmd:	STRING;
	length:	DINT;
	subStr:	STRING;
	valLen:	INT;		// Number of character for the value
END_VAR
// During INIT it might happen that the command index is 0.
// These cases should be discarded.
IF idx <= 0	THEN
	M_ReadFromReply	:= TRUE;
	RETURN;
END_IF

IF bInitCmd	THEN
	cmd		:= cfg.cmdList_Init[idx].cmd;
	length	:= cfg.cmdList_Init[idx].length;
ELSE
	cmd		:= cfg.cmdList_Read[idx].cmd;
	length	:= cfg.cmdList_Read[idx].length;
END_IF

IF length <> 0  AND  LEN(stat.sReply) <> length THEN
	stat.sErrorText	:= 'Wrong reply length';
	M_ReadFromReply	:= FALSE;
	RETURN;
END_IF

// Check if sent command was correct.
IF	FIND(stat.sReply,'NO_DEF') > 0	OR 
	FIND(stat.sReply,'_RANGE') > 0	OR 
	FIND(stat.sReply,'_LOGIC') > 0		THEN
	// Wrong command sent. This is an error.
	stat.sErrorText	:= 'Incorrect command';
	M_ReadFromReply	:= FALSE;
	RETURN;
END_IF

// Check the structure of the reply.
// Example 1 - Data query with 6 characters for the value:
//    CMD:   1 2 3 0 0 3 0 9 0 2 = ? 1 1 2 cR
//    Reply: 1 2 3 1 0 3 0 9 0 6 0 0 0 6 3 3 0 3 7 cR
//    valLen = 6 (from '06' in reply)
//    value = 633
// Example 2 - Data query with 3 characters for the value:
//    CMD:   1 2 3 0 0 0 6 0 0 2 = ? x x x cR
//    Reply: 1 2 3 1 0 0 6 0 0 3 0 0 2 y y y cR
//    valLen = 3 (from '03' in reply)
//    value = 002 = 2
// Example 3 - Command (reply is identical to command):
//    CMD:   0 4 2 1 0 0 1 0 0 6 1 1 1 1 1 1 0 2 0 cR
//    Reply: 0 4 2 1 0 0 1 0 0 6 1 1 1 1 1 1 0 2 0 cR
//    valLen = 6 (from '06' in reply)
//    value = 111111
//
// Compared to the first 10 chars of the command, 
// the reply should modify characters 3 and 9 (index starts from 0)
// reply[3] = 1
// reply[9] = length - 14
//
// So, we want to convert: 1 2 3 0 0 3 0 9 0 2
//                     to: 1 2 3 1 0 3 0 9 0 6
// Extract first 10 characters from the command
subStr	:= MID(cmd,10,1);
// Replace character [3] with '1', i.e. with ASCII 49.
subStr[3]	:= 49;
// Replace character [9] with expected number of characters in the value.
valLen	:= DINT_TO_INT(length - 14);
// Convert integer to character.
subStr[9]	:= INT_TO_BYTE(valLen + 48);	// 48 is ascii '0'.
IF	FIND(stat.sReply,subStr) <> 1	THEN
	// Wrong reply received. This is an error.
	stat.sErrorText	:= 'Wrong reply received';
	M_ReadFromReply	:= FALSE;
	RETURN;
END_IF


//
// All fine so far. Let's extract the reading.
//
// The actual reply is contained in the 'valLen' (3 or 6) characters starting 
// from char [10] (11-the character for MID() function).
subStr	:= MID(stat.sReply, valLen, 11);

// Remove the 3-character checksum from the command.
cmd	:= MID(cmd, LEN(cmd)-3,1);


IF cmd = cfg.C_CMD_sFwVersion	THEN
	stat.sFwVersion		:= MID(subStr, 6, 1);
ELSIF cmd = cfg.C_CMD_sHwVersion	THEN
	stat.sHwVersion		:= MID(subStr, 6, 1);
ELSIF cmd = cfg.C_CMD_nNominalSpeed	THEN
	stat.nNominalSpeed	:= LREAL_TO_DINT(STRING_TO_LREAL(subStr));
ELSIF cmd = cfg.C_CMD_bON	THEN
	stat.bON	:= STRING_TO_BOOL(subStr) <> FALSE;
ELSIF cmd = cfg.C_CMD_nCtrlMode	THEN
	stat.nCtrlMode	:= STRING_TO_DINT(subStr);
ELSIF cmd = cfg.C_CMD_sErrorCode	THEN
	IF	FIND(subStr,'Err') > 0	OR 
		FIND(subStr,'Wrn') > 0		THEN
		// There is an Error or Warning.
		stat.sFailureCode	:= MID(subStr, 6, 1);
		stat.bFailure		:= TRUE;
	ELSE
		stat.sFailureCode	:= 'OK';
		stat.bFailure		:= FALSE;
	END_IF
ELSIF cmd = cfg.C_CMD_bTargetSpeed	THEN
	stat.bTargetSpeed	:= STRING_TO_BOOL(subStr) <> FALSE;
ELSIF cmd = cfg.C_CMD_nMotorCurr	THEN
	stat.nMotorCurr	:= STRING_TO_DINT(subStr) * 10;	// [mA]
ELSIF cmd = cfg.C_CMD_nPumpHours	THEN
	stat.nPumpHours	:= STRING_TO_DINT(subStr);
ELSIF cmd = cfg.C_CMD_nMotorVolt	THEN
	stat.nMotorVolt	:= STRING_TO_DINT(subStr) / 100;
	stat.lrMotorVolt:= STRING_TO_LREAL(subStr) / 100.0;	// [V]
ELSIF cmd = cfg.C_CMD_nElecHours	THEN
	stat.nElecHours	:= STRING_TO_DINT(subStr);
ELSIF cmd = cfg.C_CMD_nElecTemp	THEN
	stat.nElecTemp	:= STRING_TO_DINT(subStr);
ELSIF cmd = cfg.C_CMD_nPumpTemp	THEN
	stat.nPumpTemp	:= STRING_TO_DINT(subStr);
ELSIF cmd = cfg.C_CMD_nPumpSpeed	THEN
	stat.nPumpSpeed	:= LREAL_TO_DINT(STRING_TO_LREAL(subStr));
END_IF


M_ReadFromReply	:= TRUE;	// OK
END_METHOD

METHOD M_UpdateStatus
VAR_INPUT
END_VAR
// Update Status from digital inputs readings
stat.bReady		:= i_bReady;
stat.bFailure	:= NOT i_bError;	// Active low

stat.bMoving	:= stat.bReady OR stat.nPumpSpeed > 0;

// Set Control Mode Label
(*
	1 = remote
	2 = RS-485
	4 = PV.can
	8 = Fieldbus
	16 = E74
	255 = unlock interface selection
*)
CASE stat.nCtrlMode	OF
	1:		stat.sCtrlMode	:= 'REMOTE';
	2:		stat.sCtrlMode	:= 'RS-485';
	4:		stat.sCtrlMode	:= 'PV.can';
	8:		stat.sCtrlMode	:= 'FIELDBUS';
	16:		stat.sCtrlMode	:= 'E74';
ELSE
	stat.sCtrlMode	:= 'UNKNOWN';
END_CASE
END_METHOD

END_FUNCTION_BLOCK

// POUs/Pumps/FB_CRYO_PUMP_MVP030
FUNCTION_BLOCK FB_CRYO_PUMP_MVP030 EXTENDS FB_CRYO_PUMP_SERIAL
VAR_INPUT
END_VAR
VAR_OUTPUT
END_VAR
VAR
	
	{attribute 'OPC.UA.DA' := '1'}
	cfg:		T_CRYO_PUMP_MVP030_CFG;	
	{attribute 'OPC.UA.DA' := '1'}
	ctrl:		T_CRYO_PUMP_BASE_CTRL;	
	{attribute 'OPC.UA.DA' := '1'}
	{attribute 'OPC.UA.DA.Access' := '1'}
	stat:		T_CRYO_PUMP_MVP030_STAT;	


	// Input signals
	i_bReady		AT %I*:	BOOL;	// Turbo Pump Ready (signal DO1)
	i_bError		AT %I*:	BOOL;	// If FALSE, Error present - active low (signal DO2)

	// Output signals q_bStart already defined in FB_CRYO_TMP_BASE.
	// q_bStart should activate a relay that 
	// connects Pin 7 with Pin 5 - DI Pumping station

END_VAR


// Execute the base class object FB_CRYO_PUMP_SERIAL
SUPER^();

METHOD M_Configure
VAR_INPUT
END_VAR
VAR
	//
	// List of INIT commands.
	//
	cmdList_Init_MVP030:	ARRAY [1..8] OF T_CRYO_PUMP_CMD := [
		(cmd := cfg.C_CMD_sCtrlViaInt, 		length := 17),	// Reply of 17 chars with the terminator!	
		(cmd := cfg.C_CMD_sFwVersion, 		length := 20),	
		(cmd := cfg.C_CMD_sHwVersion, 		length := 20),
		(cmd := cfg.C_CMD_nNominalSpeed,	length := 20),
		(cmd := '', 						length := 0),
		(cmd := '', 						length := 0),
		(cmd := '', 						length := 0),
		(cmd := '', 						length := 0)];

	//
	//	List of READ (and WRITE) commands.
	// NOTE: Monitoring loop stops on first cmd = ''.
	//
	cmdList_Read_MVP030:	ARRAY [1..16] OF T_CRYO_PUMP_CMD := [
		(cmd := cfg.C_CMD_bON, 				length := 20),	// Reply of 20 chars with the terminator!	
		(cmd := cfg.C_CMD_nCtrlMode, 		length := 17),	
		(cmd := cfg.C_CMD_sErrorCode, 		length := 20),
		(cmd := cfg.C_CMD_nMotorCurr, 		length := 20),
		(cmd := cfg.C_CMD_nPumpHours, 		length := 20),
		(cmd := cfg.C_CMD_nMotorVolt, 		length := 20),
		(cmd := cfg.C_CMD_nElecPower, 		length := 20),
		(cmd := cfg.C_CMD_nPumpTemp, 		length := 20),
		(cmd := cfg.C_CMD_nPumpSpeed, 		length := 20),
		(cmd := '', 						length := 0),
		(cmd := '', 						length := 0),
		(cmd := '', 						length := 0),
		(cmd := '', 						length := 0),
		(cmd := '', 						length := 0),
		(cmd := '', 						length := 0),
		(cmd := '', 						length := 0)];
	
		i:	INT;
END_VAR
IF NOT bStarted	THEN
	//
	// START: Mandatory for ALL pumps !!!
	//
	// Set references from FB_RS_BASE
	cfgRef	REF=cfg;
	ctrlRef	REF=ctrl;
	statRef	REF=stat;

	// Set references from FB_CRYO_TMP_BASE
	cfgBaseRef	REF=cfg;
	ctrlBaseRef	REF=ctrl;
	statBaseRef	REF=stat;
	
	// Copy input parameters to configuration
	cfg.nModel			:= in_nModel;
	cfg.bAutoMonitor	:= in_bAutoMonitor;
	cfg.tDelay_Periodic	:= DINT_TO_TIME(in_nPeriod);
	
	
	// Set pointers to arrays of commands
	ptrInitCmds	:= ADR(cfg.cmdList_Init);(* Pointer to INIT commands *)
	ptrReadCmds	:= ADR(cfg.cmdList_Read);(* Pointer to READ commands *)
	
	// TODO in FB that extends the functionality
	// Set pointers to comm, i.e.
	ptrCommCfg	:= ADR(comm.cfg);	(* Pointer to comm.cfg instance *)
	ptrCommCtrl	:= ADR(comm.ctrl);	(* Pointer to comm.ctrl instance *)
	ptrCommStat	:= ADR(comm.stat);	(* Pointer to comm.stat instance *)
	
	// Set comm suffixes for commands and replies
	ptrCommCfg^.sCmdSuffix		:= in_sCmdSuffix;
	ptrCommCfg^.sReplySuffix	:= in_sReplySuffix;

	statRef.bConfigured	:= TRUE;
	bStarted			:= TRUE;
	//
	// END: Mandatory for ALL pumps !!!
	//


	//
	// ATH specific configuration
	//
	
	// Assign INIT and READ commands.
	cfg.cmdList_Init	:= cmdList_Init_MVP030;
	cfg.cmdList_Read	:= cmdList_Read_MVP030;
	
	// Add checksum to all INIT and READ commands
	FOR i:=1 TO 8 DO
		IF cfg.cmdList_Init[i].cmd <> '' THEN
			cfg.cmdList_Init[i].cmd	:= M_PVP_Checksum(cfg.cmdList_Init[i].cmd);
		ELSE
			EXIT;
		END_IF
	END_FOR
	
	FOR i:=1 TO 16 DO
		IF cfg.cmdList_Read[i].cmd <> '' THEN
			cfg.cmdList_Read[i].cmd	:= M_PVP_Checksum(cfg.cmdList_Read[i].cmd);
		ELSE
			EXIT;
		END_IF
	END_FOR
	
END_IF
END_METHOD

METHOD M_GetSpeed : DINT
VAR_INPUT
END_VAR
M_GetSpeed	:= stat.nPumpSpeed;
END_METHOD

METHOD M_IsReady : BOOL
VAR_INPUT
END_VAR
M_IsReady	:= stat.bReady;
END_METHOD

METHOD M_IsRunning : BOOL
VAR_INPUT
END_VAR
M_IsRunning	:= stat.bMoving;
END_METHOD

METHOD M_ReadFromReply : BOOL
// Method to check correctness of the reply and assign the result to a status variable.
VAR_INPUT
	idx:		INT;		(* arr [idx] will hold the first extracted value, arr [idx+1] the second one, etc. *)
	bInitCmd:	BOOL := FALSE;
END_VAR
VAR
	pos:	INT;
	cmd:	STRING;
	length:	DINT;
	subStr:	STRING;
	valLen:	INT;		// Number of character for the value
END_VAR
// During INIT it might happen that the command index is 0.
// These cases should be discarded.
IF idx <= 0	THEN
	M_ReadFromReply	:= TRUE;
	RETURN;
END_IF

IF bInitCmd	THEN
	cmd		:= cfg.cmdList_Init[idx].cmd;
	length	:= cfg.cmdList_Init[idx].length;
ELSE
	cmd		:= cfg.cmdList_Read[idx].cmd;
	length	:= cfg.cmdList_Read[idx].length;
END_IF

IF length <> 0  AND  LEN(stat.sReply) <> length THEN
	stat.sErrorText	:= 'Wrong reply length';
	M_ReadFromReply	:= FALSE;
	RETURN;
END_IF

// Check if sent command was correct.
IF	FIND(stat.sReply,'NO_DEF') > 0	OR 
	FIND(stat.sReply,'_RANGE') > 0	OR 
	FIND(stat.sReply,'_LOGIC') > 0		THEN
	// Wrong command sent. This is an error.
	stat.sErrorText	:= 'Incorrect command';
	M_ReadFromReply	:= FALSE;
	RETURN;
END_IF

// Check the structure of the reply.
// Example 1 - Data query with 6 characters for the value:
//    CMD:   1 2 3 0 0 3 0 9 0 2 = ? 1 1 2 cR
//    Reply: 1 2 3 1 0 3 0 9 0 6 0 0 0 6 3 3 0 3 7 cR
//    valLen = 6 (from '06' in reply)
//    value = 633
// Example 2 - Data query with 3 characters for the value:
//    CMD:   1 2 3 0 0 0 6 0 0 2 = ? x x x cR
//    Reply: 1 2 3 1 0 0 6 0 0 3 0 0 2 y y y cR
//    valLen = 3 (from '03' in reply)
//    value = 002 = 2
// Example 3 - Command (reply is identical to command):
//    CMD:   0 4 2 1 0 0 1 0 0 6 1 1 1 1 1 1 0 2 0 cR
//    Reply: 0 4 2 1 0 0 1 0 0 6 1 1 1 1 1 1 0 2 0 cR
//    valLen = 6 (from '06' in reply)
//
// Compared to the first 10 chars of the command, 
// the reply should modify characters 3 and 9 (index starts from 0)
// reply[3] = 1
// reply[9] = length - 14
//
// So, we want to convert: 1 2 3 0 0 3 0 9 0 2
//                     to: 1 2 3 1 0 3 0 9 0 6
// Extract first 10 characters from the command
subStr	:= MID(cmd,10,1);
// Replace character [3] with '1', i.e. with ASCII 49.
subStr[3]	:= 49;
// Replace character [9] with expected number of characters in the value.
valLen	:= DINT_TO_INT(length - 14);
// Convert integer to character.
subStr[9]	:= INT_TO_BYTE(valLen + 48);
IF	FIND(stat.sReply,subStr) <> 1	THEN
	// Wrong reply received. This is an error.
	stat.sErrorText	:= 'Wrong reply received';
	M_ReadFromReply	:= FALSE;
	RETURN;
END_IF


//
// All fine so far. Let's extract the reading.
//
// The actual reply is contained in the 'valLen' (3 or 6) characters starting 
// from char [10] (11-the character for MID() function).
subStr	:= MID(stat.sReply, valLen, 11);

// Remove the 3-character checksum from the command.
cmd	:= MID(cmd, LEN(cmd)-3,1);

IF cmd = cfg.C_CMD_sFwVersion	THEN
	stat.sFwVersion		:= MID(subStr, 6, 1);
ELSIF cmd = cfg.C_CMD_sHwVersion	THEN
	stat.sHwVersion		:= MID(subStr, 6, 1);
ELSIF cmd = cfg.C_CMD_nNominalSpeed	THEN
	stat.nNominalSpeed	:= LREAL_TO_DINT(STRING_TO_LREAL(subStr));		// [rpm]
ELSIF cmd = cfg.C_CMD_bON	THEN
	stat.bON	:= STRING_TO_BOOL(subStr) <> FALSE;
ELSIF cmd = cfg.C_CMD_nCtrlMode	THEN
	stat.nCtrlMode	:= STRING_TO_DINT(subStr);
ELSIF cmd = cfg.C_CMD_sErrorCode	THEN
	IF	FIND(subStr,'Err') > 0	OR 
		FIND(subStr,'Wrn') > 0		THEN
		// There is an Error or Warning.
		stat.sFailureCode	:= MID(subStr, 6, 1);
		stat.bFailure		:= TRUE;
	ELSE
		stat.sFailureCode	:= 'OK';
		stat.bFailure		:= FALSE;
	END_IF
ELSIF cmd = cfg.C_CMD_nMotorCurr	THEN
	stat.nMotorCurr	:= STRING_TO_DINT(subStr) * 10;		// [mA]
ELSIF cmd = cfg.C_CMD_nPumpHours	THEN
	stat.nPumpHours	:= STRING_TO_DINT(subStr);
ELSIF cmd = cfg.C_CMD_nMotorVolt	THEN
	stat.nMotorVolt	:= STRING_TO_DINT(subStr) / 100;	// [V]
	stat.lrMotorVolt:= STRING_TO_LREAL(subStr) / 100.0;	// [V]
ELSIF cmd = cfg.C_CMD_nElecPower	THEN
	stat.nElecPower	:= STRING_TO_DINT(subStr);			// [W]
ELSIF cmd = cfg.C_CMD_nPumpTemp	THEN
	stat.nPumpTemp	:= STRING_TO_DINT(subStr);			// [°C]
ELSIF cmd = cfg.C_CMD_nPumpSpeed	THEN
	stat.nPumpSpeed	:= LREAL_TO_DINT(STRING_TO_LREAL(subStr));			// [rpm]
END_IF


M_ReadFromReply	:= TRUE;	// OK
END_METHOD

METHOD M_UpdateStatus
VAR_INPUT
END_VAR
// Update Status from digital inputs readings
stat.bReady		:= i_bReady;
stat.bFailure	:= NOT i_bError;	// Active low

stat.bMoving	:= stat.bReady OR stat.nPumpSpeed > 0;

// Set Control Mode Label
(*
	1 = remote
	2 = RS-485
	4 = PV.can
	32 = Keys on the front panel
*)
CASE stat.nCtrlMode	OF
	1:		stat.sCtrlMode	:= 'REMOTE';
	2:		stat.sCtrlMode	:= 'RS-485';
	4:		stat.sCtrlMode	:= 'PV.can';
	32:		stat.sCtrlMode	:= 'Keys on Front Panel';
ELSE
	stat.sCtrlMode	:= 'UNKNOWN';
END_CASE
END_METHOD

END_FUNCTION_BLOCK

// POUs/Sensors/FB_CRYO_PRESSURE
//
// This FB reads preasure using up to two PKR 250 sensors, 
// i.e. two instances of FB_CRYO_SENSOR_PKR250.
// The resulting value is a combination of values from available/valid sensors.
// Provides status of each sensor.
// For more info, see method M_SetStatus().
//
FUNCTION_BLOCK FB_CRYO_PRESSURE
VAR_INPUT
	// IMPORTANT NOTE:
	// 		It is assumed that both pressure sensors are of same type.
	//		So, all configuration parameters are same for both sensors.
	//
	{attribute 'OPC.UA.DA' := '0'}
	// Scale factors for each sensor bits -> Volt, U = raw / scale. 
	// Default for 16-bit, +-10V or 0..10V AI: 2^16/10/2 = 3276.8 bit
	in_lrBitsPerVolt_1:	LREAL := 3276.8;	// Scale factor, U = raw / scale. Default 3276.8
	{attribute 'OPC.UA.DA' := '0'}
	in_lrBitsPerVolt_2:	LREAL := 3276.8;	// Scale factor, U = raw / scale. Default 3276.8

	{attribute 'OPC.UA.DA' := '0'}
	in_nType_1:	E_CRYO_SENSOR_TYPE_PRESS	:= E_CRYO_SENSOR_TYPE_PRESS.PKR_250;
	{attribute 'OPC.UA.DA' := '0'}
	in_nType_2:	E_CRYO_SENSOR_TYPE_PRESS	:= E_CRYO_SENSOR_TYPE_PRESS.PKR_250;
	
	
	{attribute 'OPC.UA.DA' := '0'}
	in_lrLimitInVac:	LREAL := 100.0;		// Below this value, the pressure is vacuum
	{attribute 'OPC.UA.DA' := '0'}
	in_lrLimitGoodVac:	LREAL := 10.0E-4;	// Below this value, vacuum is good
	
END_VAR
VAR
	{attribute 'OPC.UA.DA' := '1'}
	Pressure1:	FB_CRYO_SENSOR_PRESSURE;
	{attribute 'OPC.UA.DA' := '1'}
	Pressure2:	FB_CRYO_SENSOR_PRESSURE;
	
	stat:		T_CRYO_PRESSURE_STATUS;	// Complete status
END_VAR

// Get status of two vacuum gauges
M_ReadSensors();

// Set the calculated vacuum pressure
M_SetStatus();

// Get status for both vacuum gauges
METHOD M_ReadSensors
VAR_INPUT
END_VAR
Pressure1(	
	in_nType			:= in_nType_1,
	in_lrBitsPerVolt	:= in_lrBitsPerVolt_1);

Pressure2(	
	in_nType			:= in_nType_2,
	in_lrBitsPerVolt	:= in_lrBitsPerVolt_2);
END_METHOD

// Calculate pressure based on the status of the two sensors
METHOD M_SetStatus
VAR_INPUT
END_VAR
VAR
	lrTmp:		LREAL;	// Temporary var
END_VAR
//
// Determine validity and calculate pressure in user units, i.e. mbar
//
IF Pressure1.stat.bValid  AND  Pressure2.stat.bValid  THEN
	// If any of the two readings are in range, the reading is in range.
	stat.bInRange	:= (Pressure1.stat.bValueInRange  OR  Pressure2.stat.bValueInRange);
	stat.bValid			:= TRUE;
	stat.bWarningSens1	:= FALSE;
	stat.bWarningSens2	:= FALSE;
	
	// Are the readings within 10% from each other
	IF Pressure2.stat.lrPressure > 0.0 THEN
		lrTmp	:= Pressure1.stat.lrPressure / Pressure2.stat.lrPressure;
	ELSE
		lrTmp	:= 0.0;	// Dummy, just to take the higher pressure.
	END_IF
	IF lrTmp > 0.9 AND lrTmp < 1.1  THEN
		// Get the average of the two
		stat.lrPressure	:= (Pressure1.stat.lrPressure + Pressure2.stat.lrPressure) / 2;
	ELSE
		// Get the higher value
		stat.lrPressure	:= MAX(Pressure1.stat.lrPressure, Pressure2.stat.lrPressure);
	END_IF
ELSIF Pressure1.stat.bValid  AND  NOT Pressure2.stat.bValid  THEN
	// Reading of one sensor is OK.
	// However, we set a warning.
	stat.bInRange		:= Pressure1.stat.bValueInRange;
	stat.bValid			:= TRUE;
	stat.bWarningSens1	:= FALSE;
	stat.bWarningSens2	:= TRUE;
	// Take the reading of the first sensor
	stat.lrPressure		:= Pressure1.stat.lrPressure;
ELSIF NOT Pressure1.stat.bValid  AND  Pressure2.stat.bValid  THEN
	// Reading of one sensor is OK.
	// However, we set a warning.
	stat.bInRange		:= Pressure2.stat.bValueInRange;
	stat.bValid			:= TRUE;
	stat.bWarningSens1	:= TRUE;
	stat.bWarningSens2	:= FALSE;
	// Take the reading of the second sensor
	stat.lrPressure		:= Pressure2.stat.lrPressure;
ELSE
	// Both readings are not valid.
	// Reading is not valid.
	stat.bInRange		:= FALSE;
	stat.bValid			:= FALSE;
	stat.bWarningSens1	:= TRUE;
	stat.bWarningSens2	:= TRUE;
	stat.lrPressure		:= 0.0;	// Dummy if reading not valid
END_IF


//
// Set vacuum state based on the pressure level
//
IF NOT stat.bValid  THEN
	stat.bInVacuum		:= FALSE;
	stat.bVacuumGood	:= FALSE;
ELSE
	// 	Check the vacuum levels
	IF stat.lrPressure < in_lrLimitGoodVac  THEN
		stat.bInVacuum		:= TRUE;
		stat.bVacuumGood	:= TRUE;
	ELSIF stat.lrPressure < in_lrLimitInVac  THEN
		stat.bInVacuum		:= TRUE;
		stat.bVacuumGood	:= FALSE;
	ELSE
		stat.bInVacuum		:= FALSE;
		stat.bVacuumGood	:= FALSE;
	END_IF
END_IF
END_METHOD

END_FUNCTION_BLOCK

// POUs/Sensors/FB_CRYO_SENSOR_PRESSURE
FUNCTION_BLOCK FB_CRYO_SENSOR_PRESSURE EXTENDS FB_CRYO_SENSOR_BASE
VAR_INPUT
	{attribute 'OPC.UA.DA' := '0'}
	in_nType:	E_CRYO_SENSOR_TYPE_PRESS;
	{attribute 'OPC.UA.DA' := '0'}
	// Scale factor bits -> Volt, U = raw / scale. 
	// Default for 16-bit, +-10V or 0..10V AI: 2^16/10/2 = 3276.8 bit
	in_lrBitsPerVolt:	LREAL := 3276.8;	// Scale factor, U = raw / scale. Default 3276.8
	{attribute 'OPC.UA.DA' := '0'}
	in_nSampleTime:		UINT := 2000;	// Time for average read sample [ms]
END_VAR
VAR_OUTPUT
END_VAR
VAR
	{attribute 'OPC.UA.DA' := '1'}
	stat:	T_CRYO_SENSOR_STATUS_PRESS;	// Complete status

	// Timers 
	{attribute 'OPC.UA.DA' := '0'}
	fbReadTimer:	TON; (* General Timeout *)

	// Misc internal vars
	{attribute 'OPC.UA.DA' := '0'}
	nCount:			UINT := 0;		// Number of effective samples
	{attribute 'OPC.UA.DA' := '0'}
	bReadStarted:	BOOL := FALSE;	// Used for initial trigger of the read timer
	{attribute 'OPC.UA.DA' := '0'}
	lrVoltageSum:	LREAL := 0.0;	// Total sum of Valid voltages during sample time.
	{attribute 'OPC.UA.DA' := '0'}
	lrVoltageAve:	LREAL := 0.0;	// Average voltage over in_nSampleTime
END_VAR

// Set references
RefStat	REF=stat;

IF NOT bReadStarted THEN
	bReadStarted	:= TRUE;
	fbReadTimer(IN:=FALSE);
END_IF
fbReadTimer(IN:=TRUE,PT:=UINT_TO_TIME(in_nSampleTime));


// Execute the base FB
SUPER^();

// Calculate pressure based on the status in input value
METHOD M_SetStatus
VAR_INPUT
END_VAR
VAR
END_VAR
// Set pressure sensor type
stat.nType	:= in_nType;

// Update validity and the pressure in user units, i.e. mbar
CASE in_nType OF
	E_CRYO_SENSOR_TYPE_PRESS.PKR_250:
		M_SetStatus_PKR_250();
	E_CRYO_SENSOR_TYPE_PRESS.PKR_360:
		M_SetStatus_PKR_360();
	E_CRYO_SENSOR_TYPE_PRESS.CMR_361:
		M_SetStatus_CMR_361();
	E_CRYO_SENSOR_TYPE_PRESS.WRG_D_NW25:
		M_SetStatus_WRG_D_NW25();
END_CASE
END_METHOD

// Calculate pressure based on the status in input value
METHOD M_SetStatus_CMR_361
VAR_INPUT
END_VAR
VAR
	// Pfeiffer CMR361 Conversion Volt -> mbar.
	// P = (U - 1) * C1 * C2 [mbar]
	// Defaults are for Pfeiffer CMR361 (note: C1 = 0.125, C2=FullScale = 1000): 
	// P = (U - 1) * 0.125 * 1000.0 = (U-1) * 125[mbar]
	
	lrVoltage:		LREAL;	
END_VAR
// Update validity and the pressure in user units, i.e. mbar.

// Sum up all valid voltages in the range (1.0..9.8V].
IF NOT stat.bInputError  AND  stat.bInputValid  AND stat.bInputActive  THEN
	// Convert bits -> Volt
	lrVoltage	:= i_nValue / in_lrBitsPerVolt;

	// If reading is (1.0..9.8V], add the voltage to the Sum
	IF lrVoltage > 1.0  AND  lrVoltage <= 9.8 THEN
		nCount			:= nCount + 1;
		lrVoltageSum	:= lrVoltageSum + lrVoltage;
	END_IF
END_IF


// If the timer has expired, calculate the average voltage/pressure.
// Also, restart timer, and reset the counter and lrVoltageSum.
IF fbReadTimer.Q THEN
	fbReadTimer(IN:=FALSE);	// Reset timer
	IF nCount > 0 THEN
		stat.lrVoltage	:= lrVoltageSum / nCount;	// Average voltage
	ELSE
		stat.lrVoltage	:= 0.0;	// Dummy voltage - error.
	END_IF
	nCount			:= 0;
	lrVoltageSum	:= 0.0;

	// Convert Volt -> Pressure [mbar]
	// Measuring range [0.1...1100mbar] = [1.0008...9.8V]
	stat.lrPressure		:= (stat.lrVoltage - 1.0) * 125.0;

	// Check the validity of the measurement.
	// < 0.4 V - ERROR, sensor problem, Underrange
	// < 1.0V - NOT Valid, Underrange
	// < 1.0008V (0.1mbar) - Valid, underrange
	//   1.0008V (0.1mbar) .. 9.8V (1100mbar) - Valid, in range
	// > 9.8V (1100mbar) - NOT Valid, Overrange
	IF stat.lrVoltage <= 0.4	THEN
		stat.bError				:= TRUE;
		stat.bValid				:= FALSE;
		stat.bValueInRange		:= FALSE;
		stat.bValueUnderrange	:= TRUE;
		stat.bValueOverrange	:= FALSE;
	ELSIF stat.lrVoltage <= 1.0	THEN
		stat.bError				:= FALSE;
		stat.bValid				:= FALSE;
		stat.bValueInRange		:= FALSE;
		stat.bValueUnderrange	:= TRUE;
		stat.bValueOverrange	:= FALSE;
	ELSIF stat.lrVoltage < 1.0008	THEN
		stat.bError				:= FALSE;
		stat.bValid				:= TRUE;
		stat.bValueInRange		:= FALSE;
		stat.bValueUnderrange	:= TRUE;
		stat.bValueOverrange	:= FALSE;
	ELSIF stat.lrVoltage <= 9.8	THEN
		stat.bError				:= FALSE;
		stat.bValid				:= TRUE;
		stat.bValueInRange		:= TRUE;
		stat.bValueUnderrange	:= FALSE;
		stat.bValueOverrange	:= FALSE;
	ELSE
		stat.bError				:= TRUE;
		stat.bValid				:= FALSE;
		stat.bValueInRange		:= FALSE;
		stat.bValueUnderrange	:= FALSE;
		stat.bValueOverrange	:= TRUE;
	END_IF

END_IF
END_METHOD

// Calculate pressure based on the status in input value
METHOD M_SetStatus_PKR_250
VAR_INPUT
END_VAR
VAR
	// Pfeiffer PKR250/251 Conversion Volt -> mbar.
	// P = 10^(C1 * U - C2).
	// Defaults are for Pfeiffer PKR250/251 (note: C1 = 1.667, C2 = d = 11.33): 
	// P = 10^(1.667 * U - 11.33)
	// Valid range for U is 1.8-8.6
	//
	
	lrVoltage:		LREAL;
END_VAR
// Update validity and the pressure in user units, i.e. mbar.

// Sum up all valid voltages in the range [1.4..9.5V].
IF NOT stat.bInputError  AND  stat.bInputValid  AND stat.bInputActive  THEN
	// Convert bits -> Volt
	lrVoltage	:= i_nValue / in_lrBitsPerVolt;

	// If reading is [1.4..9.5V], add the voltage to the Sum
	IF lrVoltage >= 1.4  AND  lrVoltage <= 9.5 THEN
		nCount			:= nCount + 1;
		lrVoltageSum	:= lrVoltageSum + lrVoltage;
	END_IF
END_IF


// If the timer has expired, calculate the average voltage/pressure.
// Also, restart timer, and reset the counter and lrVoltageSum.
IF fbReadTimer.Q THEN
	fbReadTimer(IN:=FALSE);	// Reset timer
	IF nCount > 0 THEN
		stat.lrVoltage	:= lrVoltageSum / nCount;	// Average voltage
	ELSE
		stat.lrVoltage	:= 0.0;	// Dummy voltage - error.
	END_IF
	nCount			:= 0;
	lrVoltageSum	:= 0.0;

	// Convert Volt -> Pressure [mbar]
	// Measuring range [0.1...1100mbar] = [1.0008...9.8V]
	stat.lrPressure		:= EXPT(10.0, (1.667 * stat.lrVoltage - 11.33));

	// Check the validity of the measurement.
	// < 0.5 V - ERROR, sensor problem, Underrange
	// < 1.4V (1E-09mbar)- NOT Valid, Underrange
	// < 1.76V (4E-09mbar) - Valid, underrange
	//   1.76V (4E-09mbar) .. 8.6V (1014mbar) - Valid, in range
	// < 9.5V (1014mbar) - Valid, Overrange, fixed pressure to 1014mbar
	// >= 9.5V  - NOT Valid, Overrange
	IF stat.lrVoltage <= 0.5	THEN
		stat.bError				:= TRUE;
		stat.bValid				:= FALSE;
		stat.bValueInRange		:= FALSE;
		stat.bValueUnderrange	:= TRUE;
		stat.bValueOverrange	:= FALSE;
	ELSIF stat.lrVoltage < 1.4	THEN
		stat.bError				:= FALSE;
		stat.bValid				:= FALSE;
		stat.bValueInRange		:= FALSE;
		stat.bValueUnderrange	:= TRUE;
		stat.bValueOverrange	:= FALSE;
	ELSIF stat.lrVoltage < 1.76	THEN
		stat.bError				:= FALSE;
		stat.bValid				:= TRUE;
		stat.bValueInRange		:= FALSE;
		stat.bValueUnderrange	:= TRUE;
		stat.bValueOverrange	:= FALSE;
	ELSIF stat.lrVoltage <= 8.6	THEN
		stat.bError				:= FALSE;
		stat.bValid				:= TRUE;
		stat.bValueInRange		:= TRUE;
		stat.bValueUnderrange	:= FALSE;
		stat.bValueOverrange	:= FALSE;
	ELSIF stat.lrVoltage <= 9.5	THEN
		stat.bError				:= FALSE;
		stat.bValid				:= TRUE;
		stat.bValueInRange		:= FALSE;
		stat.bValueUnderrange	:= FALSE;
		stat.bValueOverrange	:= TRUE;
		stat.lrPressure			:= 1014.0;
	ELSE
		stat.bError				:= TRUE;
		stat.bValid				:= FALSE;
		stat.bValueInRange		:= FALSE;
		stat.bValueUnderrange	:= FALSE;
		stat.bValueOverrange	:= TRUE;
	END_IF

END_IF
END_METHOD

// Calculate pressure based on the status in input value
METHOD M_SetStatus_PKR_360
VAR_INPUT
END_VAR
VAR
	// Pfeiffer PKR360 Conversion Volt -> mbar.
	// P = 10^(C1 * U - C2).
	// Defaults are for Pfeiffer PKR250/251 (note: C1 = 1.667, C2 = d = 11.33): 
	// P = 10^(1.667 * U - 11.33)
	// Valid range for U is 1.397-8.6 (up to 9.5 fixed to 1014 mbar in SW)
	//
	
	lrVoltage:		LREAL;
END_VAR
// Update validity and the pressure in user units, i.e. mbar.

// Sum up all valid voltages in the range [1.397 .. 9.5V].
IF NOT stat.bInputError  AND  stat.bInputValid  AND stat.bInputActive  THEN
	// Convert bits -> Volt
	lrVoltage	:= i_nValue / in_lrBitsPerVolt;

	// If reading is [1.4..9.5V], add the voltage to the Sum
	IF lrVoltage >= 1.397  AND  lrVoltage <= 9.5 THEN
		nCount			:= nCount + 1;
		lrVoltageSum	:= lrVoltageSum + lrVoltage;
	END_IF
END_IF


// If the timer has expired, calculate the average voltage/pressure.
// Also, restart timer, and reset the counter and lrVoltageSum.
IF fbReadTimer.Q THEN
	fbReadTimer(IN:=FALSE);	// Reset timer
	IF nCount > 0 THEN
		stat.lrVoltage	:= lrVoltageSum / nCount;	// Average voltage
	ELSE
		stat.lrVoltage	:= 0.0;	// Dummy voltage - error.
	END_IF
	nCount			:= 0;
	lrVoltageSum	:= 0.0;

	// Convert Volt -> Pressure [mbar]
	// Measuring range [0.1...1100mbar] = [1.0008...9.5V]
	stat.lrPressure		:= EXPT(10.0, (1.667 * stat.lrVoltage - 11.33));

	// Check the validity of the measurement.
	// < 1.217 V - ERROR, sensor problem, Underrange
	// < 1.397V (1E-09mbar)- NOT Valid, Underrange
	//   8.6V (4E-09mbar) .. 8.6V (1014mbar) - Valid, in range
	// < 9.5V (1014mbar) - Valid, Overrange, fixed pressure to 1014mbar
	// >= 9.5V  - NOT Valid, Overrange
	IF stat.lrVoltage <= 1.217	THEN
		stat.bError				:= TRUE;
		stat.bValid				:= FALSE;
		stat.bValueInRange		:= FALSE;
		stat.bValueUnderrange	:= TRUE;
		stat.bValueOverrange	:= FALSE;
	ELSIF stat.lrVoltage < 1.397	THEN
		stat.bError				:= FALSE;
		stat.bValid				:= FALSE;
		stat.bValueInRange		:= FALSE;
		stat.bValueUnderrange	:= TRUE;
		stat.bValueOverrange	:= FALSE;
	ELSIF stat.lrVoltage <= 8.6	THEN
		stat.bError				:= FALSE;
		stat.bValid				:= TRUE;
		stat.bValueInRange		:= TRUE;
		stat.bValueUnderrange	:= FALSE;
		stat.bValueOverrange	:= FALSE;
	ELSIF stat.lrVoltage <= 9.5	THEN
		stat.bError				:= FALSE;
		stat.bValid				:= TRUE;
		stat.bValueInRange		:= FALSE;
		stat.bValueUnderrange	:= FALSE;
		stat.bValueOverrange	:= TRUE;
		stat.lrPressure			:= 1014.0;
	ELSE
		stat.bError				:= TRUE;
		stat.bValid				:= FALSE;
		stat.bValueInRange		:= FALSE;
		stat.bValueUnderrange	:= FALSE;
		stat.bValueOverrange	:= TRUE;
	END_IF

END_IF
END_METHOD

// Calculate pressure based on the status in input value
METHOD M_SetStatus_WRG_D_NW25
VAR_INPUT
END_VAR
VAR
	// Edwards WRG-D-NW25 Conversion Volt -> mbar.
	// Range 10^-9 .. 100
	// P = 10^(C1 * U - C2).
	// P = 10^(1.5 * U - 12.0)
	// Valid range for U is 2.0-10.0
	//
	
	lrVoltage:		LREAL;
END_VAR
// Update validity and the pressure in user units, i.e. mbar.

// Sum up all valid voltages in the range [2.0..10.0V].
IF NOT stat.bInputError  AND  stat.bInputValid  AND stat.bInputActive  THEN
	// Convert bits -> Volt
	lrVoltage	:= i_nValue / in_lrBitsPerVolt;

	// If reading is [2.0..10.0V], add the voltage to the Sum
	IF lrVoltage >= 2.0  AND  lrVoltage <= 10.0 THEN
		nCount			:= nCount + 1;
		lrVoltageSum	:= lrVoltageSum + lrVoltage;
	END_IF
END_IF


// If the timer has expired, calculate the average voltage/pressure.
// Also, restart timer, and reset the counter and lrVoltageSum.
IF fbReadTimer.Q THEN
	fbReadTimer(IN:=FALSE);	// Reset timer
	IF nCount > 0 THEN
		stat.lrVoltage	:= lrVoltageSum / nCount;	// Average voltage
	ELSE
		stat.lrVoltage	:= 0.0;	// Dummy voltage - error.
	END_IF
	nCount			:= 0;
	lrVoltageSum	:= 0.0;

	// Convert Volt -> Pressure [mbar]
	// Measuring range [0.1...1000mbar] = [2.0...10.0V]
	stat.lrPressure		:= EXPT(10.0, (1.5 * stat.lrVoltage - 12.0));

	// Check the validity of the measurement.
	// < 1.5 V - ERROR, sensor problem, Underrange
	// < 2.0V (1E-09mbar)- NOT Valid, Underrange
	// < 10.0V (1000mbar) - Valid
	// < 10.15V (1678mbar) - NOT Valid, Overrange
	// >= 10.15V  - Error, Overrange
	IF stat.lrVoltage < 1.5	THEN
		stat.bError				:= TRUE;
		stat.bValid				:= FALSE;
		stat.bValueInRange		:= FALSE;
		stat.bValueUnderrange	:= TRUE;
		stat.bValueOverrange	:= FALSE;
	ELSIF stat.lrVoltage < 2.0	THEN
		stat.bError				:= FALSE;
		stat.bValid				:= FALSE;
		stat.bValueInRange		:= FALSE;
		stat.bValueUnderrange	:= TRUE;
		stat.bValueOverrange	:= FALSE;
	ELSIF stat.lrVoltage <= 10.0	THEN
		stat.bError				:= FALSE;
		stat.bValid				:= TRUE;
		stat.bValueInRange		:= TRUE;
		stat.bValueUnderrange	:= FALSE;
		stat.bValueOverrange	:= FALSE;
	ELSIF stat.lrVoltage <= 10.15	THEN
		stat.bError				:= FALSE;
		stat.bValid				:= FALSE;
		stat.bValueInRange		:= FALSE;
		stat.bValueUnderrange	:= FALSE;
		stat.bValueOverrange	:= TRUE;
	ELSE
		stat.bError				:= TRUE;
		stat.bValid				:= FALSE;
		stat.bValueInRange		:= FALSE;
		stat.bValueUnderrange	:= FALSE;
		stat.bValueOverrange	:= TRUE;
	END_IF

END_IF
END_METHOD

END_FUNCTION_BLOCK

// POUs/Sensors/FB_CRYO_SENSOR_BASE
FUNCTION_BLOCK FB_CRYO_SENSOR_BASE
VAR_INPUT
END_VAR
VAR
	{attribute 'OPC.UA.DA' := '0'}
	i_nStatus	AT %I*: UINT;
	{attribute 'OPC.UA.DA' := '0'}
	i_nValue	AT%I*:	INT;
	
	{attribute 'OPC.UA.DA' := '0'}
	bStarted:		BOOL := FALSE;
	{attribute 'OPC.UA.DA' := '0'}
	toggleTimer:	TON;		// Timer for PDO (alive) toggle
	{attribute 'OPC.UA.DA' := '0'}
	toggleTrig:		R_TRIG;		// PDO (alive) toggle detection
	
	RefStat: 	REFERENCE TO T_CRYO_SENSOR_STATUS;
END_VAR

// Get the raw reading and the status of the input channel
M_ReadSensor();

// Calculate value and validity
M_SetStatus();

// Get input channel status and the raw reading
METHOD M_ReadSensor
VAR_INPUT
END_VAR
// Get input channel status
RefStat.bInputUnder	:= (i_nStatus AND 2#0000_0000_0000_0001) <> 0;
RefStat.bInputOver	:= (i_nStatus AND 2#0000_0000_0000_0010) <> 0;
RefStat.bInputError	:= (i_nStatus AND 2#0000_0000_0100_0000) <> 0;
RefStat.bInputToggle:= (i_nStatus AND 2#1000_0000_0000_0000) <> 0;
RefStat.bInputValid	:= (i_nStatus AND 2#0100_0000_0000_0000)  = 0;	// 0 -> PDO OK

// Get the raw reading
RefStat.nRawValue	:= i_nValue;

//
// Check if the terminal is alive.
// Start the time that will expire in 3 sec.
// If bToggle bit triggers before the timer expires, 
// this is the sign that the terminal is alive.
//
IF NOT bStarted THEN
	bStarted	:= TRUE;
	toggleTimer(IN:=FALSE);
END_IF
toggleTimer(IN:=TRUE,PT:=T#3S);
toggleTrig(CLK:=RefStat.bInputToggle);

IF toggleTrig.Q THEN
	// bToggle bit has triggered. Terminal is alive.
	RefStat.bInputActive	:= TRUE;
	// Restart the timer
	toggleTimer(IN:=FALSE);
ELSIF toggleTimer.Q THEN
	// bInputToggle bit has not triggered within 3 sec. Terminal is NOT alive.
	RefStat.bInputActive	:= FALSE;
	// Restart the timer
	toggleTimer(IN:=FALSE);
END_IF
END_METHOD

METHOD M_SetStatus
VAR_INPUT
END_VAR
// TODO USER: Implement the method.
END_METHOD

END_FUNCTION_BLOCK

// POUs/Sensors/FB_CRYO_PRESSURE_VOTE
//
// This FB calculates resulting pressure applying the selected voting method.
// Up to five pressure sensors are used in the calculation.
// The resulting value is a combination of values from available/valid sensors.
// For more info, see method M_SetStatus().
//
FUNCTION_BLOCK FB_CRYO_PRESSURE_VOTE
VAR_INPUT
	{attribute 'OPC.UA.DA' := '0'}
	in_bSimulation:	BOOL	:= FALSE;	// If TRUE, the pressure value is simulated.
	
	{attribute 'OPC.UA.DA' := '0'}
	in_nNumSensor:	INT;				// Number of sensors used by voiting method.
	
	{attribute 'OPC.UA.DA' := '0'}
	in_nVoteMethod:	E_CRYO_VOTE	:= E_CRYO_VOTE.V_AVE;	// Active voting method.
	
	// Five pointers to instances of FB_CRYO_SENSOR_PRESSURE.
	// Pointers should only be set to existing pressure sensors.
	{attribute 'OPC.UA.DA' := '0'}
	in_pSensor1:		POINTER TO FB_CRYO_SENSOR_PRESSURE	:= 0;
	{attribute 'OPC.UA.DA' := '0'}
	in_pSensor2:		POINTER TO FB_CRYO_SENSOR_PRESSURE	:= 0;
	{attribute 'OPC.UA.DA' := '0'}
	in_pSensor3:		POINTER TO FB_CRYO_SENSOR_PRESSURE	:= 0;
	{attribute 'OPC.UA.DA' := '0'}
	in_pSensor4:		POINTER TO FB_CRYO_SENSOR_PRESSURE	:= 0;
	{attribute 'OPC.UA.DA' := '0'}
	in_pSensor5:		POINTER TO FB_CRYO_SENSOR_PRESSURE	:= 0;

END_VAR
VAR
	{attribute 'OPC.UA.DA' := '1'}
	stat:		T_CRYO_PRESSURE_VOTE_STATUS;	// Complete status
	
	pSensor:	ARRAY [1..5] OF POINTER TO FB_CRYO_SENSOR_PRESSURE;
END_VAR

// If not configured yet, return.
IF NOT M_Configure()	THEN
	RETURN;
END_IF

// Set warnings for sensors with problems
M_CheckWarnings();

// Set the calculated vacuum pressure
M_SetStatus();

METHOD M_CheckWarnings : BOOL
VAR_INPUT
END_VAR
VAR
	i:			INT;
END_VAR
FOR i:=1 TO in_nNumSensor DO
	IF pSensor[i] <> 0  THEN
		// The set pointer (<> 0) indicates that the sensor is connected.
		// Warnings could be set only for connected sensors.
		IF  pSensor[i]^.stat.bValid	THEN
			// Clear warning
			M_SetWarning(i, FALSE);
		ELSE
			// Set warning
			M_SetWarning(i, TRUE);
		END_IF
	ELSE
		// Not connected sensors don't have warnings
		M_SetWarning(i, FALSE);
	END_IF
END_FOR
END_METHOD

METHOD M_Configure : BOOL
VAR_INPUT
END_VAR
VAR
	j:					INT;
END_VAR
VAR_INST
	{attribute 'OPC.UA.DA' := '0'}
	i:	INT := 0;
	{attribute 'OPC.UA.DA' := '0'}
	bConfigured:	BOOL := FALSE;
END_VAR
// The number of sensors must be between 1 and 5.
IF in_nNumSensor < 1 OR in_nNumSensor > 5 THEN
	// Set error string
	stat.sStatus	:= 'ERROR: Number of sensors (var in_nNumSensor) is not in range [1..5]';
	RETURN;
END_IF

// Configure the system in stages after boot-up.
// WARNING:
// It seems that setting of pointers takes some time and cannot be done in FB_Init.
// After 40 cycles, we set pointers to sensors.
// After 80 cycles, we set general configuration parameters and complete configuration.
IF NOT bConfigured THEN
	i	:= i + 1;
	IF i = 40 THEN
		// Assign pointers to the sensor device instances
		pSensor[1] := in_pSensor1;
		pSensor[2] := in_pSensor2;
		pSensor[3] := in_pSensor3;
		pSensor[4] := in_pSensor4;
		pSensor[5] := in_pSensor5;
	ELSIF i >= 80 THEN
		FOR j := 1 TO in_nNumSensor DO
			IF pSensor[j] <> 0 THEN
				// Set the status flag that the sensor is connected.
				M_SetConnected(j, TRUE);
				// At least one pointer is not zero.
				// We have finished configuration.
				bConfigured	:= TRUE;
			ELSE
				M_SetConnected(j, FALSE);
			END_IF
		END_FOR
	END_IF
END_IF

M_Configure	:= bConfigured;
END_METHOD

METHOD M_SetConnected : BOOL
VAR_INPUT
	in_nIndex:		INT;
	in_bConnected:	BOOL;
END_VAR
CASE in_nIndex OF
	1:
		stat.bConnSens1	:= in_bConnected;
	2:
		stat.bConnSens2	:= in_bConnected;
	3:
		stat.bConnSens3	:= in_bConnected;
	4:
		stat.bConnSens4	:= in_bConnected;
	5:
		stat.bConnSens5	:= in_bConnected;
END_CASE
END_METHOD

// Calculate pressure based on the status of the two sensors
METHOD M_SetStatus
VAR_INPUT
END_VAR
VAR
	lrTmp:		LREAL;	// Temporary var
	nSample:	INT;
	i:			INT;
END_VAR
//
// If simulated, set the simulated value and return.
//
IF in_bSimulation THEN
	stat.bSimulated	:= TRUE;
	stat.bValid		:= TRUE;
	stat.lrPressure	:= stat.lrSimPressure;
	RETURN;
ELSE
	stat.bSimulated	:= FALSE;
END_IF


//
// Get the pressure depending on the voting method.
//
CASE in_nVoteMethod OF
	E_CRYO_VOTE.V_AVE:
		M_SetStatus_Average();
	E_CRYO_VOTE.V_MIN:
		M_SetStatus_Minimum();
	E_CRYO_VOTE.V_MAX:
		M_SetStatus_Maximum();
	E_CRYO_VOTE.V_1oo2:
		M_SetStatus_FirstValid();
	E_CRYO_VOTE.V_2oo3:
		M_SetStatus_XooY(2,3);
	E_CRYO_VOTE.V_3oo5:
		M_SetStatus_XooY(3,5);
ELSE
	;
END_CASE


//
// If the reading is valid, set the simulated value to it.
// This way, switching from normal to simulation will result in
// no jump in the value.
//
IF stat.bValid  THEN
	stat.lrSimPressure	:= stat.lrPressure;
END_IF
END_METHOD

// Calculate pressure based on the average of all valid sensor readings
METHOD M_SetStatus_Average
VAR_INPUT
END_VAR
VAR
	lrTmp:		LREAL;	// Temporary var for sum of pressures
	nSample:	INT;	// Number of valid sensor readings
	i:			INT;
END_VAR
lrTmp	:= 0.0;
nSample	:= 0;
FOR i:=1 TO in_nNumSensor DO
	IF pSensor[i] <> 0  THEN
		IF  pSensor[i]^.stat.bValid	THEN
			lrTmp	:= lrTmp + pSensor[i]^.stat.lrPressure;
			nSample	:= nSample + 1;
		END_IF
	END_IF
END_FOR
IF nSample > 0	THEN
	stat.lrPressure	:= lrTmp / nSample;
	stat.bValid		:= TRUE;
ELSE
	stat.lrPressure	:= 9999;
	stat.bValid		:= FALSE;
END_IF
END_METHOD

// Calculate pressure based on the first measured valid value
METHOD M_SetStatus_FirstValid
VAR_INPUT
END_VAR
VAR
	lrTmp:		LREAL;	// Temporary var for sum of pressures
	nSample:	INT;	// Number of valid sensor readings
	i:			INT;
END_VAR
nSample	:= 0;
FOR i:=1 TO in_nNumSensor DO
	IF pSensor[i] <> 0  THEN
		IF  pSensor[i]^.stat.bValid	THEN
			lrTmp	:= pSensor[i]^.stat.lrPressure;
			nSample	:= nSample + 1;
			EXIT;
		END_IF
	END_IF
END_FOR
IF nSample > 0	THEN
	stat.lrPressure	:= lrTmp;
	stat.bValid		:= TRUE;
ELSE
	stat.lrPressure	:= 9999;
	stat.bValid		:= FALSE;
END_IF
END_METHOD

// Calculate pressure based on the highest measured valid value
METHOD M_SetStatus_Maximum
VAR_INPUT
END_VAR
VAR
	lrTmp:		LREAL;	// Temporary var for sum of pressures
	nSample:	INT;	// Number of valid sensor readings
	i:			INT;
END_VAR
lrTmp	:= -100000.0;	// Dummy starting value
nSample	:= 0;
FOR i:=1 TO in_nNumSensor DO
	IF pSensor[i] <> 0  THEN
		IF  pSensor[i]^.stat.bValid	THEN
			IF pSensor[i]^.stat.lrPressure > lrTmp THEN
				lrTmp	:= pSensor[i]^.stat.lrPressure;
			END_IF
			nSample	:= nSample + 1;
		END_IF
	END_IF
END_FOR
IF nSample > 0	THEN
	stat.lrPressure	:= lrTmp;
	stat.bValid		:= TRUE;
ELSE
	stat.lrPressure	:= 9999;
	stat.bValid		:= FALSE;
END_IF
END_METHOD

// Calculate pressure based on the lowest measured valid value
METHOD M_SetStatus_Minimum
VAR_INPUT
END_VAR
VAR
	lrTmp:		LREAL;	// Temporary var for sum of pressures
	nSample:	INT;	// Number of valid sensor readings
	i:			INT;
END_VAR
lrTmp	:= 100000.0;	// Dummy starting value
nSample	:= 0;
FOR i:=1 TO in_nNumSensor DO
	IF pSensor[i] <> 0  THEN
		IF  pSensor[i]^.stat.bValid	THEN
			IF pSensor[i]^.stat.lrPressure < lrTmp THEN
				lrTmp	:= pSensor[i]^.stat.lrPressure;
			END_IF
			nSample	:= nSample + 1;
		END_IF
	END_IF
END_FOR
IF nSample > 0	THEN
	stat.lrPressure	:= lrTmp;
	stat.bValid		:= TRUE;
ELSE
	stat.lrPressure	:= 9999;
	stat.bValid		:= FALSE;
END_IF
END_METHOD

// Calculate pressure based on the status of the two sensors
METHOD M_SetStatus_XooY
VAR_INPUT
	in_nNum:	INT;	// Number of readings to select for voting (X)
	in_nTotal:	INT;	// Total number of readings to check (Y)
END_VAR
VAR
	idx_i, idx_j:	INT;
	nTmp:		INT;			// Temporary INT var
	lrTmp:		LREAL	:= 0.0;	// Temporary var for sum of pressures
	nValid:		INT		:= 0;	// Total number of valid readings
	nSample:	INT		:= 0;	// Number of valid sensor readings
	
	aDiff:		ARRAY [1..5,1..5] OF LREAL;	// Table of absolute differences
	aDiffSum:	ARRAY [1..5] OF LREAL;		// Array of sums of absolute differences
	// Array of indexes of sums of absolute differences
	aDiffSumIdx:ARRAY [1..5] OF INT := [1,2,3,4,5];		
	lrAbsDiff:	LREAL;						// Absolute difference between two readings
	
	i:			INT;
	j:			INT;
END_VAR
//
//	Get the number of valid readings and calculate the average
//
FOR i:=1 TO in_nTotal DO
	IF pSensor[i] <> 0  THEN
		IF  pSensor[i]^.stat.bValid	THEN
			lrTmp	:= lrTmp + pSensor[i]^.stat.lrPressure;
			nValid	:= nValid + 1;
		END_IF
	END_IF
END_FOR


//
// Vote X out of Y
//
IF nValid >= in_nNum	THEN
	//
	// Calculate relative differences between two readings, 
	// relative to the bigger ABS value.
	// Table is symetric. Calculate only the half (triangle) on the right. 
	// Make a copy to the other half.
	//
	FOR i:=1 TO in_nTotal DO
		FOR j:=i+1 TO in_nTotal DO
			IF pSensor[i] <> 0  AND  pSensor[j] <> 0	THEN
				IF pSensor[i]^.stat.bValid  AND  pSensor[j]^.stat.bValid	THEN
					lrAbsDiff	:= ABS(pSensor[i]^.stat.lrPressure - pSensor[j]^.stat.lrPressure);
					aDiff[i,j]	:= lrAbsDiff;
					aDiff[j,i]	:= lrAbsDiff;
				ELSE
					aDiff[i,j]	:= 9999.0;
					aDiff[j,i]	:= 9999.0;
				END_IF
			ELSE
				aDiff[i,j]	:= 9999.0;
				aDiff[j,i]	:= 9999.0;
			END_IF
		END_FOR
	END_FOR

	//
	// Get the sum of all differences for each reading.
	//
	FOR i:=1 TO in_nTotal DO
		aDiffSum[i]	:= 0.0;
		FOR j:=1 TO in_nTotal DO
			aDiffSum[i]	:= aDiffSum[i] + aDiff[i,j];
		END_FOR
	END_FOR

	//
	// Sort the indexes for differences in accending order (low sum first).
	//
	FOR i:=1 TO in_nTotal DO
		FOR j:=i+1 TO in_nTotal DO
			idx_i	:= aDiffSumIdx[i];
			idx_j	:= aDiffSumIdx[j];
			IF aDiffSum[idx_j] < aDiffSum[idx_i]	THEN
				// Swap indexes
				nTmp			:= aDiffSumIdx[j];
				aDiffSumIdx[j]	:= aDiffSumIdx[i];
				aDiffSumIdx[i]	:= nTmp;
			END_IF
		END_FOR
	END_FOR

	
	//					
	// Get the average of selected in_nNum readings.
	// Assign the result to the pressure.
	//
	lrTmp	:= 0.0;
	FOR i:=1 TO in_nNum DO
		idx_i	:= aDiffSumIdx[i];
		lrTmp	:= lrTmp + pSensor[idx_i]^.stat.lrPressure;
	END_FOR
	
	stat.lrPressure	:= lrTmp / in_nNum;
	stat.bValid		:= TRUE;
ELSE
	stat.lrPressure	:= 9999;
	stat.bValid		:= FALSE;
END_IF
END_METHOD

METHOD M_SetWarning : BOOL
VAR_INPUT
	in_nIndex:		INT;
	in_bWarning:	BOOL;
END_VAR
CASE in_nIndex OF
	1:
		stat.bWarnSens1	:= in_bWarning;
	2:
		stat.bWarnSens2	:= in_bWarning;
	3:
		stat.bWarnSens3	:= in_bWarning;
	4:
		stat.bWarnSens4	:= in_bWarning;
	5:
		stat.bWarnSens5	:= in_bWarning;
END_CASE
END_METHOD

END_FUNCTION_BLOCK

// POUs/Sensors/FB_CRYO_SBG232
FUNCTION_BLOCK FB_CRYO_SBG232
VAR_INPUT
	in_sName:		string	   := 'IO-Link SBG232';
	in_sUnitFlow:	STRING(16) := 'L/min';	//	Units for Flow, default [L/min] 
	in_sUnitTemp:	STRING(16) := '°C';		//	Units for Temperature, default [°C] 
END_VAR
VAR_OUTPUT
END_VAR
VAR
	//
	// Variables to be linked
	//
	
	// InfoData -> State of IO-Link master, e.g. EL6224.
	i_nCouplerState			AT %I*:	UINT;	
	// DeviceState Inputs -> State Ch# of IO-Link master, e.g. EL6224.
	i_nDeviceStateInputCh	AT %I*:	USINT;	
	// Raw device data: IO-Link Port# -> Port#:process data
	i_ArrPortProcessData	AT %I*:	ARRAY [0..3] OF USINT;
	
	
	stat:	T_CRYO_SBG232_STAT;
	
END_VAR

// Configure if it hasn't been done.
M_Configure();

// Extract sensor reading from the raw value.
M_UpdateStatus();

METHOD M_Configure
VAR_INPUT
END_VAR
IF NOT stat.bConfigured	THEN
	stat.bConfigured	:= TRUE;
	
	stat.sName			:= in_sName;
	
	stat.flow.sUnits	:= in_sUnitFlow;
	stat.temp.sUnits	:= in_sUnitTemp;

	stat.flow.sType		:= 'Flow';
	stat.temp.sType		:= 'Temperature';

END_IF
END_METHOD

METHOD M_SetError
VAR_INPUT
	nSensor:	E_CRYO_SBG232_SENSOR_TYPE;
	sError:		STRING;
END_VAR
VAR
	refSensor:	REFERENCE TO T_CRYO_IOLINK_SENSOR_STATUS;
END_VAR
IF nSensor	= E_CRYO_SBG232_SENSOR_TYPE.FLOW	THEN
	refSensor	REF=stat.flow;
ELSIF nSensor	= E_CRYO_SBG232_SENSOR_TYPE.TEMP	THEN
	refSensor	REF=stat.temp;
END_IF

refSensor.bError		:= TRUE;
refSensor.bInRange		:= FALSE;
refSensor.bValid		:= FALSE;
refSensor.sStatus		:= sError;
END_METHOD

METHOD M_SetReading
VAR_INPUT
	nSensor:	E_CRYO_SBG232_SENSOR_TYPE;
	lrValue:	LREAL;
END_VAR
VAR
	refSensor:	REFERENCE TO T_CRYO_IOLINK_SENSOR_STATUS;
END_VAR
IF nSensor	= E_CRYO_SBG232_SENSOR_TYPE.FLOW	THEN
	refSensor	REF=stat.flow;
ELSIF nSensor	= E_CRYO_SBG232_SENSOR_TYPE.TEMP	THEN
	refSensor	REF=stat.temp;
END_IF

refSensor.bOverrange	:= FALSE;
refSensor.bUnderrange	:= FALSE;
refSensor.bError		:= FALSE;
refSensor.bInRange		:= TRUE;
refSensor.bValid		:= TRUE;
refSensor.lrValue		:= lrValue;
refSensor.sStatus		:= 'OK';
END_METHOD

METHOD M_UpdateStatus
VAR_INPUT
END_VAR
VAR
	lrVal:	LREAL;
END_VAR
// General check if the EL6224 and IO-Link are OK.
IF i_nCouplerState	<> 8	THEN
	stat.sStatus	:= 'IO-Link terminal not in OP state. Check the mapping.';
	M_SetError(E_CRYO_SBG232_SENSOR_TYPE.FLOW, 'IO-Link terminal not in OP state');
	M_SetError(E_CRYO_SBG232_SENSOR_TYPE.TEMP, 'IO-Link terminal not in OP state');
	RETURN;
ELSIF i_nDeviceStateInputCh	<> 3	THEN
	stat.sStatus	:= 'IO-Link Channel not in OP state';
	M_SetError(E_CRYO_SBG232_SENSOR_TYPE.FLOW, 'IO-Link Channel not in OP state');
	M_SetError(E_CRYO_SBG232_SENSOR_TYPE.TEMP, 'IO-Link Channel not in OP state');
	RETURN;
ELSE
	stat.sStatus	:= 'OK';
END_IF


//////////////
// Flow
//////////////

lrVal	:= (256.0 * i_ArrPortProcessData[0] + i_ArrPortProcessData[1]) / 100.0;
stat.flow.lrValue	:= lrVal;

IF lrVal = 18.05	THEN
	stat.flow.bOverrange	:= TRUE;
	stat.flow.bUnderrange	:= FALSE;
	M_SetError(E_CRYO_SBG232_SENSOR_TYPE.FLOW, 'Overrange');
ELSE
	M_SetReading(E_CRYO_SBG232_SENSOR_TYPE.FLOW, lrVal);
END_IF


////////////////
// Temperature
////////////////

lrVal	:= TRUNC(256.0 * i_ArrPortProcessData[2] + i_ArrPortProcessData[3]) / 4;	// /4 = SHR(2)
stat.temp.lrValue	:= lrVal;


IF lrVal = 123.0	THEN
	stat.temp.bOverrange	:= TRUE;
	stat.temp.bUnderrange	:= FALSE;
	M_SetError(E_CRYO_SBG232_SENSOR_TYPE.TEMP, 'Overrange');
ELSIF lrVal = -33.0	THEN
	stat.temp.bOverrange	:= FALSE;
	stat.temp.bUnderrange	:= TRUE;
	M_SetError(E_CRYO_SBG232_SENSOR_TYPE.TEMP, 'Underrange');
ELSE
	M_SetReading(E_CRYO_SBG232_SENSOR_TYPE.TEMP, lrVal);
END_IF
END_METHOD

END_FUNCTION_BLOCK

// POUs/Sensors/FB_CRYO_SENSOR_TEMPERATURE
FUNCTION_BLOCK FB_CRYO_SENSOR_TEMPERATURE EXTENDS FB_CRYO_SENSOR_BASE
VAR_INPUT
	{attribute 'OPC.UA.DA' := '0'}
	in_nType:				E_CRYO_SENSOR_TYPE_TEMP	:= E_CRYO_SENSOR_TYPE_TEMP.PT100;
	{attribute 'OPC.UA.DA' := '0'}
	in_lrScale:				LREAL := 0.1;		// Scale factor, T = raw * scale. Default 0.1
	{attribute 'OPC.UA.DA' := '0'}
	in_bIgnoreUnderrange:	BOOL  := FALSE;		// If T, underrange will be treated as bValid.
	{attribute 'OPC.UA.DA' := '0'}
	in_nRampPeriodSec:		UDINT := 60;		// Ramp measurement period [sec]. Default 60 sec.
	// If true, temperature calculated from measured resistance.
	// With this flag active, temperature range is extended to -240 degC.
	{attribute 'OPC.UA.DA' := '0'}
	in_bResistor_1_64:		BOOL := FALSE;		
END_VAR
VAR_OUTPUT
END_VAR
VAR
	{attribute 'OPC.UA.DA' := '1'}
	stat:	T_CRYO_SENSOR_STATUS_TEMP;	// Complete status

	{attribute 'OPC.UA.DA' := '0'}
	bRampTimerStarted:	BOOL := FALSE;
	{attribute 'OPC.UA.DA' := '0'}
	rampTimer:	TON;		// Timer for calculating ramp
	
	// Lookup table when converting resistance to Celsius, range [-240..200].
	// NOTE: RTD Element in CoE of the RTD terminal, e.g., EL3201
	//       must be configured for "Resistor 1/64 Ohm..."
	//       Also, in_bResistor_1_64 must be set to TRUE.
	LookupTable:	ARRAY [0..88] OF T_CRYO_PT100_OHM2C_REC := [
			(celsius := 	-240.0	, ohm := 	0.911	),
			(celsius := 	-235.0	, ohm := 	3.150	),
			(celsius := 	-230.0	, ohm := 	5.377	),
			(celsius := 	-225.0	, ohm := 	7.594	),
			(celsius := 	-220.0	, ohm := 	9.799	),
			(celsius := 	-215.0	, ohm := 	11.995	),
			(celsius := 	-210.0	, ohm := 	14.180	),
			(celsius := 	-205.0	, ohm := 	16.356	),
			(celsius := 	-200.0	, ohm := 	18.522	),
			(celsius := 	-195.0	, ohm := 	20.679	),
			(celsius := 	-190.0	, ohm := 	22.827	),
			(celsius := 	-185.0	, ohm := 	24.967	),
			(celsius := 	-180.0	, ohm := 	27.098	),
			(celsius := 	-175.0	, ohm := 	29.221	),
			(celsius := 	-170.0	, ohm := 	31.336	),
			(celsius := 	-165.0	, ohm := 	33.444	),
			(celsius := 	-160.0	, ohm := 	35.545	),
			(celsius := 	-155.0	, ohm := 	37.638	),
			(celsius := 	-150.0	, ohm := 	39.724	),
			(celsius := 	-145.0	, ohm := 	41.804	),
			(celsius := 	-140.0	, ohm := 	43.877	),
			(celsius := 	-135.0	, ohm := 	45.945	),
			(celsius := 	-130.0	, ohm := 	48.006	),
			(celsius := 	-125.0	, ohm := 	50.061	),
			(celsius := 	-120.0	, ohm := 	52.110	),
			(celsius := 	-115.0	, ohm := 	54.155	),
			(celsius := 	-110.0	, ohm := 	56.194	),
			(celsius := 	-105.0	, ohm := 	58.227	),
			(celsius := 	-100.0	, ohm := 	60.256	),
			(celsius := 	-95.0	, ohm := 	62.280	),
			(celsius := 	-90.0	, ohm := 	64.300	),
			(celsius := 	-85.0	, ohm := 	66.315	),
			(celsius := 	-80.0	, ohm := 	68.326	),
			(celsius := 	-75.0	, ohm := 	70.332	),
			(celsius := 	-70.0	, ohm := 	72.335	),
			(celsius := 	-65.0	, ohm := 	74.333	),
			(celsius := 	-60.0	, ohm := 	76.328	),
			(celsius := 	-55.0	, ohm := 	78.319	),
			(celsius := 	-50.0	, ohm := 	80.306	),
			(celsius := 	-45.0	, ohm := 	82.290	),
			(celsius := 	-40.0	, ohm := 	84.271	),
			(celsius := 	-35.0	, ohm := 	86.248	),
			(celsius := 	-30.0	, ohm := 	88.222	),
			(celsius := 	-25.0	, ohm := 	90.192	),
			(celsius := 	-20.0	, ohm := 	92.160	),
			(celsius := 	-15.0	, ohm := 	94.124	),
			(celsius := 	-10.0	, ohm := 	96.086	),
			(celsius := 	-5.0	, ohm := 	98.044	),
			(celsius := 	0.0		, ohm := 	100.000	),
			(celsius := 	5.0		, ohm := 	101.953	),
			(celsius := 	10.0	, ohm := 	103.903	),
			(celsius := 	15.0	, ohm := 	105.850	),
			(celsius := 	20.0	, ohm := 	107.794	),
			(celsius := 	25.0	, ohm := 	109.735	),
			(celsius := 	30.0	, ohm := 	111.674	),
			(celsius := 	35.0	, ohm := 	113.610	),
			(celsius := 	40.0	, ohm := 	115.542	),
			(celsius := 	45.0	, ohm := 	117.473	),
			(celsius := 	50.0	, ohm := 	119.400	),
			(celsius := 	55.0	, ohm := 	121.324	),
			(celsius := 	60.0	, ohm := 	123.246	),
			(celsius := 	65.0	, ohm := 	125.164	),
			(celsius := 	70.0	, ohm := 	127.080	),
			(celsius := 	75.0	, ohm := 	128.992	),
			(celsius := 	80.0	, ohm := 	130.901	),
			(celsius := 	85.0	, ohm := 	132.808	),
			(celsius := 	90.0	, ohm := 	134.710	),
			(celsius := 	95.0	, ohm := 	136.610	),
			(celsius := 	100.0	, ohm := 	138.506	),
			(celsius := 	105.0	, ohm := 	140.399	),
			(celsius := 	110.0	, ohm := 	142.288	),
			(celsius := 	115.0	, ohm := 	144.173	),
			(celsius := 	120.0	, ohm := 	146.054	),
			(celsius := 	125.0	, ohm := 	147.932	),
			(celsius := 	130.0	, ohm := 	149.805	),
			(celsius := 	135.0	, ohm := 	151.674	),
			(celsius := 	140.0	, ohm := 	153.539	),
			(celsius := 	145.0	, ohm := 	155.400	),
			(celsius := 	150.0	, ohm := 	157.256	),
			(celsius := 	155.0	, ohm := 	159.107	),
			(celsius := 	160.0	, ohm := 	160.953	),
			(celsius := 	165.0	, ohm := 	162.794	),
			(celsius := 	170.0	, ohm := 	164.630	),
			(celsius := 	175.0	, ohm := 	166.460	),
			(celsius := 	180.0	, ohm := 	168.285	),
			(celsius := 	185.0	, ohm := 	170.104	),
			(celsius := 	190.0	, ohm := 	171.917	),
			(celsius := 	195.0	, ohm := 	173.723	),
			(celsius := 	200.0	, ohm := 	175.523	)];

			lrTemStep:	LREAL	:= 5.0; 	// Temperature step in the table.
			nLastIndex:	INT		:= 0;

END_VAR

// Set references
RefStat	REF=stat;

// Execute the base FB
SUPER^();

// Calculate Temperature change ramp
M_GetRamp();

METHOD M_GetRamp
VAR_INPUT
END_VAR
VAR_INST
	{attribute 'OPC.UA.DA' := '0'}
	lrRampStartTempK:	LREAL;	// Temperature at start of ramp timer [K]
END_VAR
VAR
	nRampPeriodSec:		UDINT;	// Ramp measurement period [sec].
END_VAR
IF NOT bRampTimerStarted THEN
	bRampTimerStarted	:= TRUE;
	lrRampStartTempK	:= stat.lrTempK;
	rampTimer(IN:=FALSE);
END_IF

// Execute timer.
// Ramp measurement period should be > 0
nRampPeriodSec	:= in_nRampPeriodSec;
IF nRampPeriodSec = 0 THEN
	nRampPeriodSec	:= 60;
END_IF
rampTimer(IN:=TRUE,PT:=UDINT_TO_TIME(nRampPeriodSec)*1000);

// Calculate ramp at time expiry
IF rampTimer.Q THEN
	// Calculate the temperature ramp per minute
	IF stat.bValid THEN
		stat.lrRamp	:= (stat.lrTempK - lrRampStartTempK) * 60.0 / nRampPeriodSec;
	ELSE
		stat.lrRamp	:= 0.0;
	END_IF

	// Current temperature is the starting value of the ramp
	lrRampStartTempK	:= stat.lrTempK;

	// Restart the timer
	rampTimer(IN:=FALSE);
END_IF
END_METHOD

METHOD M_PT100_Interpolate_Ohm2C : LREAL
VAR_INPUT
	in_lrOhm:	LREAL;	// Resistance reading [Ohm]
	// Index of the first lookup table entry with 
	// value lower than the measured resistance.
	in_nIndex:	INT;	
END_VAR
VAR
	lrR1, lrR2:	LREAL;	// Temporary variables
END_VAR
IF in_nIndex = 0 OR in_nIndex = 88	THEN
	M_PT100_Interpolate_Ohm2C	:= LookupTable[in_nIndex].celsius;
ELSE
	// Linear interpolation Example
	//	Index 8		(celsius := 	-200.0	, ohm := 	18.522	),
	//  Reading                               ohm := 	20.123
	//	Index 9		(celsius := 	-195.0	, ohm := 	20.679	),
	//
	//   TempC = -200.0 + (20.123-18.522) / (20.679-18.522) * 5.0 
	//         = -200.0 + 1.601 / 2.157 * 5.0
	//         = -196.289 degC

	lrR1	:= in_lrOhm - LookupTable[in_nIndex].ohm;
	lrR2	:= LookupTable[in_nIndex+1].ohm - LookupTable[in_nIndex].ohm;
	M_PT100_Interpolate_Ohm2C	:= LookupTable[in_nIndex].celsius + lrR1/lrR2 * lrTemStep;
END_IF
END_METHOD

// Convert raw resistance reading [bit] (Ohm*64) to degrees Celsius.
// The input value has to be devided by 64 to get the reading in [Ohm].
METHOD M_PT100_Ohm2C : LREAL
VAR_INPUT
	in_lrOhmRaw:	INT;	// Raw reading [bit]. [Ohm] = in_lrOhmRaw/64
END_VAR
VAR
	i:		INT;
	lrOhm:	LREAL; 	// PT100 Resistance reading [Ohm]
END_VAR
// Raw reading of -1 means a broken wire or failed sensor.
// The convention is to return 850 degC
IF in_lrOhmRaw	= -1	THEN
	M_PT100_Ohm2C	:= 850.0;
	RETURN;
END_IF

// Get reading in [Ohm]
lrOhm	:= INT_TO_LREAL(in_lrOhmRaw) / 64.0;


// Find the first index in the table
// where the resistance value is lower that the reading.

IF lrOhm > LookupTable[nLastIndex].ohm	THEN
	// We are increasing the index until we find a reading in the
	// table that is higher than the measurement
	FOR i := nLastIndex TO 88	DO
		IF i = 88	THEN
			// We are at the highest temperature in the lookup table.
			// Take that value;
			M_PT100_Ohm2C	:= LookupTable[i].celsius;
			RETURN;
		ELSE
			IF lrOhm < LookupTable[i].ohm	THEN
				// We crossed the correct reading.
				// Remember the index for faster next reading.
				nLastIndex	:= i-1;
				IF nLastIndex < 0	THEN
					nLastIndex	:= 0;
				END_IF
				M_PT100_Ohm2C	:= M_PT100_Interpolate_Ohm2C(lrOhm,nLastIndex);
				RETURN;
			ELSIF lrOhm = LookupTable[i].ohm	THEN
				// We crossed the correct reading.
				// Remember the index for faster next reading.
				nLastIndex	:= i;
				M_PT100_Ohm2C	:= M_PT100_Interpolate_Ohm2C(lrOhm,nLastIndex);
				RETURN;
			END_IF
		END_IF
	END_FOR
ELSIF lrOhm < LookupTable[nLastIndex].ohm	THEN
	// We are decreasing the index until we find a reading in the
	// table that is higher than the measurement
	FOR i := nLastIndex TO 0 BY  -1	DO
		IF i <= 0	THEN
			// We are at the lowest temperature in the lookup table.
			// Take that value;
			M_PT100_Ohm2C	:= LookupTable[0].celsius;
			RETURN;
		ELSE
			IF lrOhm > LookupTable[i].ohm	THEN
				// We crossed the correct reading.
				// Remember the index for faster next reading.
				nLastIndex	:= i;
				M_PT100_Ohm2C	:= M_PT100_Interpolate_Ohm2C(lrOhm,nLastIndex);
				RETURN;
			ELSIF lrOhm = LookupTable[i].ohm	THEN
				// We crossed the correct reading.
				// Remember the index for faster next reading.
				nLastIndex	:= i;
				M_PT100_Ohm2C	:= M_PT100_Interpolate_Ohm2C(lrOhm,nLastIndex);
				RETURN;
			END_IF
		END_IF
	END_FOR
ELSE
	M_PT100_Ohm2C	:= M_PT100_Interpolate_Ohm2C(lrOhm,nLastIndex);
	RETURN;
END_IF
END_METHOD

// Calculate pressure based on the status in input value
METHOD M_SetStatus
VAR_INPUT
END_VAR
VAR
END_VAR
// Set temperature sensor type
stat.nType	:= in_nType;

// Update value depending on the sensor type.
// So far, only PT100 supported.
CASE in_nType OF
	E_CRYO_SENSOR_TYPE_TEMP.PT100:
		M_SetStatus_PT100();
END_CASE
END_METHOD

// Calculate pressure based on the status in input value
METHOD M_SetStatus_PT100
VAR_INPUT
END_VAR
VAR
END_VAR
//
// Set the temperature as it is read.
// Later on we decide if it is valid or not.
//
IF NOT in_bResistor_1_64	THEN
	// Standard RTD reading
	stat.lrTempC	:= i_nValue * in_lrScale;	// Set temperature in deg C
	stat.lrTempK	:= stat.lrTempC + 273.15;	// Set temperature in deg K
ELSE	
	// RTD reading of resistance.
	// i_nValue is in [Ohm]
	stat.lrTempC	:= M_PT100_Ohm2C(i_nValue);	// Set temperature in deg C
	stat.lrTempK	:= stat.lrTempC + 273.15;	// Set temperature in deg K
END_IF

// Reading in Celsius of 850.0 means an error.
// In this case, set the Kelvin reading to 850.0 as well.
// Set error and not Valid and return.
IF stat.lrTempC = 850.0	THEN
	stat.lrTempK	:= 850.0;
	stat.bError		:= TRUE;
	stat.bValid		:= FALSE;
	RETURN;
END_IF

//
// Update validity
// Note: bInputError = (bInputUnder OR bInputOver)
//       bValid      = TRUE if PDO is OK (nothing to do with bError)
//
IF stat.bInputActive THEN
	IF stat.bInputError  AND  stat.bInputUnder  AND  in_bIgnoreUnderrange 	THEN
		// Sometimes we ignore underrange because PT100 cannot read below -200C.
		// The bUnderrange flag is still active!!!
		stat.bError	:= FALSE;
		stat.bValid	:= TRUE;
	ELSIF stat.bInputError 	THEN
		stat.bError	:= TRUE;
		stat.bValid	:= FALSE;
	ELSE
		stat.bError	:= FALSE;
		stat.bValid	:= TRUE;
	END_IF
ELSE
	stat.bError	:= TRUE;
	stat.bValid	:= FALSE;
END_IF
END_METHOD

END_FUNCTION_BLOCK

// POUs/Sensors/FB_CRYO_TEMPERATURE
//
// This FB reads temperature using up to two sensors, i.e. instances of FB_CRYO_PT100.
// The resulting value is the temperature of the first available/valid sensor.
// Provides status of each sensor.
//
FUNCTION_BLOCK FB_CRYO_TEMPERATURE
VAR_INPUT
	{attribute 'OPC.UA.DA' := '0'}
	in_bSimulation:	BOOL	:= FALSE;	// If TRUE, the temperature value is simulated.
	
	{attribute 'OPC.UA.DA' := '0'}
	in_nType_1:				E_CRYO_SENSOR_TYPE_TEMP	:= E_CRYO_SENSOR_TYPE_TEMP.PT100;
	{attribute 'OPC.UA.DA' := '0'}
	in_nType_2:				E_CRYO_SENSOR_TYPE_TEMP	:= E_CRYO_SENSOR_TYPE_TEMP.PT100;
	{attribute 'OPC.UA.DA' := '0'}
	in_lrScale_1:			LREAL := 0.1;	// Scale factor, T = raw * scale. Default 0.1
	{attribute 'OPC.UA.DA' := '0'}
	in_lrScale_2:			LREAL := 0.1;	// Scale factor, T = raw * scale. Default 0.1
	{attribute 'OPC.UA.DA' := '0'}
	in_bIgnoreUnderrange_1:	BOOL := TRUE;	// If True, underrange is also valid
	{attribute 'OPC.UA.DA' := '0'}
	in_bIgnoreUnderrange_2:	BOOL := TRUE;	// If True, underrange is also valid
	{attribute 'OPC.UA.DA' := '0'}
	in_nRampPeriodSec:		UDINT := 60;	// Ramp measurement period [sec]. Default 60 sec.
	
END_VAR
VAR
	{attribute 'OPC.UA.DA' := '1'}
	Temperature1:	FB_CRYO_SENSOR_TEMPERATURE;
	{attribute 'OPC.UA.DA' := '1'}
	Temperature2:	FB_CRYO_SENSOR_TEMPERATURE;
	
	{attribute 'OPC.UA.DA' := '1'}
	stat:			T_CRYO_TEMPERATURE_STATUS;
END_VAR

// Get the raw reading and the status of the input channel
M_ReadSensors();

// Calculate temperatures and validity
M_SetStatus();

METHOD M_GetTemperatureFromLakeshore
VAR_INPUT
	bValid:		BOOL;	// Flag if reading is valid
	lrTempK:	LREAL;	// Lakeshore reading in degK 
	lrTempC:	LREAL;	// Lakeshore reading in degC 
END_VAR
//
// Check if the temperature is coming from the simulator 
// of the Lakeshore temperature.
//
// The simulator reading is always valid.
// If the temperature is not linked to a simulator,
// it will not be Valid since it is not mapped at all!!!
// If simulated, Temperature1 has to be linked to the simulator.
// Temperature2 should not be used/mapped in that case.
//
IF	Temperature1.stat.bValid THEN
	// Temperature is coming from a simulator.
	stat.bValid 		:= TRUE;
	stat.bWarningSens1	:= FALSE;
	stat.bWarningSens2	:= FALSE;
	stat.lrTempK		:= Temperature1.stat.lrTempK;
	stat.lrTempC		:= Temperature1.stat.lrTempC;
ELSIF bValid THEN
	// Temperature is coming from Lakeshore and is Valid.
	stat.bValid 		:= TRUE;
	stat.bWarningSens1	:= FALSE;
	stat.bWarningSens2	:= FALSE;
	stat.lrTempK		:= lrTempK;
	stat.lrTempC		:= lrTempC;
ELSE
	// Temperature is coming from Lakeshore and is NOT Valid.
	stat.bValid 		:= FALSE;
	stat.bWarningSens1	:= TRUE;
	stat.bWarningSens2	:= TRUE;
	stat.lrTempK		:= 850.0;
	stat.lrTempC		:= 850.0;
END_IF
END_METHOD

// Get input channel status and the raw reading
METHOD M_ReadSensors
VAR_INPUT
END_VAR
Temperature1(	in_nType				:= in_nType_1,
				in_lrScale 				:= in_lrScale_1, 
				in_bIgnoreUnderrange	:= in_bIgnoreUnderrange_1,
				in_nRampPeriodSec		:= in_nRampPeriodSec);

Temperature2(	in_nType				:= in_nType_2,
				in_lrScale 				:= in_lrScale_2, 
				in_bIgnoreUnderrange	:= in_bIgnoreUnderrange_2,
				in_nRampPeriodSec		:= in_nRampPeriodSec);
END_METHOD

METHOD M_SetStatus
VAR_INPUT
END_VAR
VAR
	lrTmp:		LREAL;	// Temporary var
END_VAR
//
// If simulated, set the simulated value and return.
// Note: Simulated temperature is in [K] !!!
//
IF in_bSimulation THEN
	stat.bSimulated	:= TRUE;
	stat.bValid		:= TRUE;
	stat.lrTempK	:= stat.lrSimTempK;
	stat.lrTempC	:= stat.lrSimTempK - 273.15;
	RETURN;
ELSE
	stat.bSimulated	:= FALSE;
END_IF


//
// Determine validity and calculate temperature in degC and degK
//
IF Temperature1.stat.bValid  AND  Temperature2.stat.bValid  THEN
	// Reading is OK.
	stat.bValid			:= TRUE;
	stat.bWarningSens1	:= FALSE;
	stat.bWarningSens2	:= FALSE;

	// Take the reading of the first sensor if it is not underrange
	// or both readings are underrange.
	IF	NOT Temperature1.stat.bInputUnder	OR
		(Temperature1.stat.bInputUnder  AND  Temperature2.stat.bInputUnder) THEN
		// T1 - NOT underrange  OR  both underrange
		// Take T1
		stat.lrRamp		:= Temperature1.stat.lrRamp;
		stat.lrTempC	:= Temperature1.stat.lrTempC;
		stat.lrTempK	:= Temperature1.stat.lrTempK;
		stat.bInRange	:= NOT Temperature1.stat.bInputUnder;
	ELSE
		// T1 - underrange
		// T2 - NOT underrange
		// Take T2
		stat.lrRamp		:= Temperature2.stat.lrRamp;
		stat.lrTempC	:= Temperature2.stat.lrTempC;
		stat.lrTempK	:= Temperature2.stat.lrTempK;
		stat.bInRange	:= NOT Temperature2.stat.bInputUnder;
	END_IF
	
ELSIF Temperature1.stat.bValid  AND  NOT Temperature2.stat.bValid  THEN
	// Reading of sensor #1 is OK.
	// However, we set a warning for sensor #2.
	stat.bValid			:= TRUE;
	stat.bWarningSens1	:= FALSE;
	stat.bWarningSens2	:= TRUE;
	// Take the reading of the first sensor
	stat.lrRamp			:= Temperature1.stat.lrRamp;
	stat.lrTempC		:= Temperature1.stat.lrTempC;
	stat.lrTempK		:= Temperature1.stat.lrTempK;
	stat.bInRange		:= NOT Temperature1.stat.bInputUnder;
	
ELSIF NOT Temperature1.stat.bValid  AND  Temperature2.stat.bValid  THEN
	// Reading of sensor #1 is NOT OK.
	// Reading of sensor #2 is OK.
	// However, we set a warning.
	stat.bValid			:= TRUE;
	stat.bWarningSens1	:= TRUE;
	stat.bWarningSens2	:= FALSE;
	// Take the reading of the second sensor
	stat.lrRamp			:= Temperature2.stat.lrRamp;
	stat.lrTempC		:= Temperature2.stat.lrTempC;
	stat.lrTempK		:= Temperature2.stat.lrTempK;
	stat.bInRange		:= NOT Temperature2.stat.bInputUnder;
	
ELSE
	// Both readings are not valid.
	// Reading is not valid.
	stat.bInRange		:= FALSE;
	stat.bValid			:= FALSE;
	stat.bWarningSens1	:= TRUE;
	stat.bWarningSens2	:= TRUE;
	// Readings are not valid.
	// The value is not important.
	// Take the value of the first sensor.
	// It might show under/over range.
	stat.lrRamp			:= 0.0;
	stat.lrTempC		:= Temperature1.stat.lrTempC;
	stat.lrTempK		:= Temperature1.stat.lrTempK;

END_IF


//
// If the reading is valid, set the simulated value to it.
// This way, switching from normal to simulation will result in
// no jump in the value.
//
IF stat.bValid  THEN
	stat.lrSimTempK	:= stat.lrTempK;
END_IF
END_METHOD

END_FUNCTION_BLOCK

// POUs/Simulation/FB_CRYO_SIM_CTRL
FUNCTION_BLOCK FB_CRYO_SIM_CTRL
VAR_INPUT
	in_ptr_Cryo_Ctrl:	POINTER TO FB_CRYO_CTRL;
END_VAR
VAR
	{attribute 'OPC.UA.DA' := '1'}
	SIM_Temp_Mirror:		FB_CRYO_SIM_TEMPERATURE;

	{attribute 'OPC.UA.DA' := '1'}
	SIM_Temp_LN2_Exhaust:	FB_CRYO_SIM_TEMPERATURE;
	
	{attribute 'OPC.UA.DA' := '1'}
	SIM_Temp_LN2_Inlet:		FB_CRYO_SIM_TEMPERATURE;
	
	{attribute 'OPC.UA.DA' := '1'}
	SIM_Temp_DET:			FB_CRYO_SIM_TEMPERATURE;
	
	{attribute 'OPC.UA.DA' := '1'}
	SIM_Pressure_Cryo:	FB_CRYO_SIM_PRESSURE;		// Cryo Pressure simulator
	
	{attribute 'OPC.UA.DA' := '1'}
	SIM_Pressure_Evac:	FB_CRYO_SIM_PRESSURE;		// Evacuation Pressure simulator
	
	
	
	{attribute 'OPC.UA.DA' := '1'}
	nCryoState:		E_CRYO_CTRL_STATE	:= E_CRYO_CTRL_STATE.NONE;
	{attribute 'OPC.UA.DA' := '0'}
	nCryoOldState:	E_CRYO_CTRL_STATE	:= E_CRYO_CTRL_STATE.NONE;
	
	{attribute 'OPC.UA.DA' := '0'}
	trgCMD:			R_TRIG;
	{attribute 'OPC.UA.DA' := '0'}
	trgEvacOn:		R_TRIG;
	{attribute 'OPC.UA.DA' := '0'}
	trgEvacOff:		F_TRIG;
	{attribute 'OPC.UA.DA' := '0'}
	trgInVacuum:	R_TRIG;
	{attribute 'OPC.UA.DA' := '0'}
	trgPrecoolOff:	F_TRIG;
	{attribute 'OPC.UA.DA' := '0'}
	trgCoolOff:		F_TRIG;
	{attribute 'OPC.UA.DA' := '0'}
	trgWarmupOff:	F_TRIG;
	
	nRampPeriod:	UDINT := 20000;
	
	{attribute 'OPC.UA.DA' := '0'}
	lrTmp:	LREAL;
	
	
END_VAR

//
// Get Cryo controller State
//
nCryoState	:= in_ptr_Cryo_Ctrl^.stat.nState;


//
// Execute simulators for all temperatures and pressures, etc.
//
SIM_Temp_Mirror(
	in_lrScale		:= in_ptr_Cryo_Ctrl^.Temp_Mirror.in_lrScale_1, 
	in_lrTempK		:= );
	
SIM_Temp_LN2_Exhaust(
	in_lrScale		:= in_ptr_Cryo_Ctrl^.Temp_LN2_Exhaust.in_lrScale_1, 
	in_lrTempK		:= 88.75,	//	Variation 88.75 +- 11.25, i.e. [77.50..100.00]
	in_lrTempDelta	:= 11.25,
	in_nPeriod		:= 10000,
	in_bAutoSine	:= TRUE);
	
SIM_Temp_LN2_Inlet(
	in_lrScale		:= in_ptr_Cryo_Ctrl^.Temp_LN2_Inlet.in_lrScale_1, 
	in_lrTempK		:= 77.15);
	
SIM_Temp_DET(
	in_lrScale		:= in_ptr_Cryo_Ctrl^.Temp_DET.in_lrScale_1, 
	in_lrTempK		:= );
	
SIM_Pressure_Cryo(
	in_nType		:= in_ptr_Cryo_Ctrl^.Pressure_Cryo.in_nType_1,
	in_lrBitsPerVolt:= in_ptr_Cryo_Ctrl^.Pressure_Cryo.in_lrBitsPerVolt_1, 
	in_nPeriod		:= nRampPeriod);
	
SIM_Pressure_Evac(
	in_nType		:= in_ptr_Cryo_Ctrl^.Pressure_Evac.in_nType_1,
	in_lrBitsPerVolt:= in_ptr_Cryo_Ctrl^.Pressure_Evac.in_lrBitsPerVolt_1, 
	in_nPeriod		:= nRampPeriod);


	
	
//	
// Capture Cryo controller change of state.
//
trgCMD(CLK:=(nCryoState<>nCryoOldState));
nCryoOldState	:= nCryoState;

// NOTE: This code is execute only once on each State change.
IF trgCMD.Q  THEN
	// The state of Cryo controller has changed.
	// Take action with simulators.
	CASE nCryoState OF
		
		/////////////////////////////////
		E_CRYO_CTRL_STATE.PRE_COOLING:
		/////////////////////////////////
		//
		// Trigger Bench temperature ramp 1 K below PRE_COOL threshold
		SIM_Temp_Mirror.M_RampTo(
			in_lrValueEnd	:= in_ptr_Cryo_Ctrl^.cfg.lrTemp_Precooled-1.0,
			in_nPeriod		:= nRampPeriod);

		// Trigger DET temperature ramp 1 K below PRE_COOL threshold.
		// Slow down the ramp compared to the Bench, so
		// DET temperature is slightly higher during cooldown.
		// The final temperature is the same as for the Bench.
		SIM_Temp_DET.M_RampTo(
			in_lrValueEnd	:= in_ptr_Cryo_Ctrl^.cfg.lrTemp_Precooled-1.0,
			in_nPeriod		:= nRampPeriod + 5000);
			
		/////////////////////////////////
		E_CRYO_CTRL_STATE.COOLING_DOWN:
		/////////////////////////////////
		//
		// Trigger temperature ramp 1 K below COOL threshold
		SIM_Temp_Mirror.M_RampTo(
			in_lrValueEnd	:= in_ptr_Cryo_Ctrl^.cfg.lrTemp_Cold-1.0,
			in_nPeriod		:= nRampPeriod);
			
		// Trigger temperature ramp 1 K below COOL threshold
		// Slow down the ramp compared to the Bench, so
		// DET temperature is slightly higher during cooldown.
		// The final temperature is the same as for the Bench.
		SIM_Temp_DET.M_RampTo(
			in_lrValueEnd	:= in_ptr_Cryo_Ctrl^.cfg.lrTemp_Cold-1.0,
			in_nPeriod		:= nRampPeriod + 5000);
			
